LIN {X 0,Y 524.233,Z 362.321,A -85,B 0,C 180,E1 -4759.475,E2 -4759.475} C_VEL
LIN {X 0,Y 524.045,Z 370.841,A -85,B 0,C 180,E1 -4760.349,E2 -4760.349} C_VEL
LIN {X 0,Y 523.843,Z 378.7,A -85,B 0,C 180,E1 -4761.319,E2 -4761.319} C_VEL
LIN {X 0,Y 523.623,Z 386.372,A -85,B 0,C 180,E1 -4762.48,E2 -4762.48} C_VEL
LIN {X 0,Y 523.511,Z 393.443,A -85,B 0,C 180,E1 -4763.834,E2 -4763.834} C_VEL
LIN {X 0,Y 523.384,Z 398.145,A -85,B 0,C 180,E1 -4764.993,E2 -4764.993} C_VEL
LIN {X 0,Y 523.443,Z 401.738,A -85,B 0,C 180,E1 -4766.15,E2 -4766.15} C_VEL
LIN {X 0,Y 523.367,Z 403.59,A -85,B 0,C 180,E1 -4766.921,E2 -4766.921} C_VEL
LIN {X 0,Y 523.335,Z 404.979,A -85,B 0,C 180,E1 -4767.691,E2 -4767.691} C_VEL
LIN {X 0,Y 523.25,Z 406.574,A -85,B 0,C 180,E1 -4769.23,E2 -4769.23} C_VEL
LIN {X 0,Y 523.247,Z 406.79,A -85,B 0,C 180,E1 -4770,E2 -4770} C_VEL
LIN {X 0,Y 523.274,Z 405.972,A -85,B 0,C 180,E1 -4771.539,E2 -4771.539} C_VEL
LIN {X 0,Y 523.335,Z 404.983,A -85,B 0,C 180,E1 -4772.309,E2 -4772.309} C_VEL
LIN {X 0,Y 523.367,Z 403.595,A -85,B 0,C 180,E1 -4773.079,E2 -4773.079} C_VEL
LIN {X 0,Y 523.423,Z 400.675,A -85,B 0,C 180,E1 -4774.235,E2 -4774.235} C_VEL
LIN {X 0,Y 523.461,Z 396.72,A -85,B 0,C 180,E1 -4775.392,E2 -4775.392} C_VEL
LIN {X 0,Y 523.519,Z 391.508,A -85,B 0,C 180,E1 -4776.577,E2 -4776.577} C_VEL
LIN {X 0,Y 523.645,Z 385.219,A -85,B 0,C 180,E1 -4777.713,E2 -4777.713} C_VEL
LIN {X 0,Y 523.835,Z 377.219,A -85,B 0,C 180,E1 -4778.875,E2 -4778.875} C_VEL
LIN {X 0,Y 524.06,Z 369.064,A -85,B 0,C 180,E1 -4779.845,E2 -4779.845} C_VEL
LIN {X 0,Y 524.345,Z 359.117,A -85,B 0,C 180,E1 -4780.815,E2 -4780.815} C_VEL
LIN {X 0,Y 524.633,Z 347.823,A -85,B 0,C 180,E1 -4781.693,E2 -4781.693} C_VEL
LIN {X 0,Y 524.915,Z 336.875,A -85,B 0,C 180,E1 -4782.369,E2 -4782.369} C_VEL
LIN {X 0,Y 525.16,Z 324.67,A -85,B 0,C 180,E1 -4782.953,E2 -4782.953} C_VEL
LIN {X 0,Y 525.409,Z 311.875,A -85,B 0,C 180,E1 -4783.389,E2 -4783.389} C_VEL
LIN {X 0,Y 525.572,Z 298.314,A -85,B 0,C 180,E1 -4783.681,E2 -4783.681} C_VEL
LIN {X 0,Y 525.831,Z 204.563,A -85,B 0,C 180,E1 -4784.972,E2 -4784.972} C_VEL
LIN {X 0,Y 524.293,Z 195.105,A -85,B 0,C 180,E1 -4785.172,E2 -4785.172} C_VEL
LIN {X 0,Y 524.444,Z 184.228,A -85,B 0,C 180,E1 -4786.945,E2 -4786.945} C_VEL
LIN {X 0,Y 524.807,Z 168.725,A -85,B 0,C 180,E1 -4789.559,E2 -4789.559} C_VEL
LIN {X 0,Y 525.149,Z 155.599,A -85,B 0,C 180,E1 -4791.799,E2 -4791.799} C_VEL
LIN {X 0,Y 523.95,Z 148.335,A -85,B 0,C 180,E1 -4793.152,E2 -4793.152} C_VEL
LIN {X 0,Y 523.928,Z 148.217,A -85,B 0,C 180,E1 -4796.273,E2 -4796.273} C_VEL
LIN {X 0,Y 523.949,Z 148.223,A -85,B 0,C 180,E1 -4799.322,E2 -4799.322} C_VEL
LIN {X 0,Y 523.929,Z 148.219,A -85,B 0,C 180,E1 -4802.449,E2 -4802.449} C_VEL
LIN {X 0,Y 523.913,Z 148.227,A -85,B 0,C 180,E1 -4805.226,E2 -4805.226} C_VEL
LIN {X 0,Y 523.908,Z 148.214,A -85,B 0,C 180,E1 -4808.101,E2 -4808.101} C_VEL
LIN {X 0,Y 523.912,Z 148.228,A -85,B 0,C 180,E1 -4811.093,E2 -4811.093} C_VEL
LIN {X 0,Y 523.927,Z 148.218,A -85,B 0,C 180,E1 -4814.228,E2 -4814.228} C_VEL
LIN {X 0,Y 523.909,Z 148.224,A -85,B 0,C 180,E1 -4816.832,E2 -4816.832} C_VEL
LIN {X 0,Y 523.93,Z 148.224,A -85,B 0,C 180,E1 -4818.907,E2 -4818.907} C_VEL
LIN {X 0,Y 523.905,Z 148.215,A -85,B 0,C 180,E1 -4821.897,E2 -4821.897} C_VEL
LIN {X 0,Y 523.919,Z 148.218,A -85,B 0,C 180,E1 -4824.91,E2 -4824.91} C_VEL
LIN {X 0,Y 523.924,Z 148.219,A -85,B 0,C 180,E1 -4827.679,E2 -4827.679} C_VEL
LIN {X 0,Y 523.941,Z 148.22,A -85,B 0,C 180,E1 -4830.676,E2 -4830.676} C_VEL
LIN {X 0,Y 523.961,Z 148.213,A -85,B 0,C 180,E1 -4833.728,E2 -4833.728} C_VEL
LIN {X 0,Y 523.9,Z 148.219,A -85,B 0,C 180,E1 -4836.269,E2 -4836.269} C_VEL
LIN {X 0,Y 523.933,Z 148.225,A -85,B 0,C 180,E1 -4838.766,E2 -4838.766} C_VEL
LIN {X 0,Y 523.937,Z 148.215,A -85,B 0,C 180,E1 -4841.22,E2 -4841.22} C_VEL
LIN {X 0,Y 523.918,Z 148.217,A -85,B 0,C 180,E1 -4843.638,E2 -4843.638} C_VEL
LIN {X 0,Y 523.924,Z 148.219,A -85,B 0,C 180,E1 -4846.028,E2 -4846.028} C_VEL
LIN {X 0,Y 524,Z 148.208,A -85,B 0,C 180,E1 -4849.177,E2 -4849.177} C_VEL
LIN {X 0,Y 524.013,Z 148.211,A -85,B 0,C 180,E1 -4852.292,E2 -4852.292} C_VEL
LIN {X 0,Y 524.066,Z 148.203,A -85,B 0,C 180,E1 -4854.614,E2 -4854.614} C_VEL
LIN {X 0,Y 524.093,Z 148.196,A -85,B 0,C 180,E1 -4857.694,E2 -4857.694} C_VEL
LIN {X 0,Y 524.113,Z 148.196,A -85,B 0,C 180,E1 -4860.768,E2 -4860.768} C_VEL
LIN {X 0,Y 524.059,Z 148.2,A -85,B 0,C 180,E1 -4863.075,E2 -4863.075} C_VEL
LIN {X 0,Y 524.022,Z 148.21,A -85,B 0,C 180,E1 -4866.159,E2 -4866.159} C_VEL
LIN {X 0,Y 523.991,Z 148.212,A -85,B 0,C 180,E1 -4868.484,E2 -4868.484} C_VEL
LIN {X 0,Y 523.991,Z 148.21,A -85,B 0,C 180,E1 -4871.741,E2 -4871.741} C_VEL
LIN {X 0,Y 523.98,Z 148.208,A -85,B 0,C 180,E1 -4875.053,E2 -4875.053} C_VEL
LIN {X 0,Y 523.952,Z 148.217,A -85,B 0,C 180,E1 -4877.97,E2 -4877.97} C_VEL
LIN {X 0,Y 523.961,Z 148.218,A -85,B 0,C 180,E1 -4880.411,E2 -4880.411} C_VEL
LIN {X 0,Y 523.908,Z 148.219,A -85,B 0,C 180,E1 -4882.894,E2 -4882.894} C_VEL
LIN {X 0,Y 523.941,Z 148.216,A -85,B 0,C 180,E1 -4885.419,E2 -4885.419} C_VEL
LIN {X 0,Y 523.96,Z 148.218,A -85,B 0,C 180,E1 -4888,E2 -4888} C_VEL
LIN {X 0,Y 523.934,Z 148.217,A -85,B 0,C 180,E1 -4890.856,E2 -4890.856} C_VEL
LIN {X 0,Y 523.951,Z 148.215,A -85,B 0,C 180,E1 -4893.736,E2 -4893.736} C_VEL
LIN {X 0,Y 523.911,Z 148.219,A -85,B 0,C 180,E1 -4896.405,E2 -4896.405} C_VEL
LIN {X 0,Y 523.912,Z 148.219,A -85,B 0,C 180,E1 -4899.086,E2 -4899.086} C_VEL
LIN {X 0,Y 523.949,Z 148.215,A -85,B 0,C 180,E1 -4902.119,E2 -4902.119} C_VEL
LIN {X 0,Y 523.937,Z 148.215,A -85,B 0,C 180,E1 -4905.311,E2 -4905.311} C_VEL
LIN {X 0,Y 523.909,Z 148.22,A -85,B 0,C 180,E1 -4906.932,E2 -4906.932} C_VEL
LIN {X 0,Y 523.246,Z 148.308,A -85,B 0,C 180,E1 -4907.574,E2 -4907.574} C_VEL
LIN {X 0,Y 520.405,Z 148.661,A -85,B 0,C 180,E1 -4908.616,E2 -4908.616} C_VEL
LIN {X 0,Y 517.999,Z 148.961,A -85,B 0,C 180,E1 -4909.455,E2 -4909.455} C_VEL
LIN {X 0,Y 516.962,Z 149.086,A -85,B 0,C 180,E1 -4910.103,E2 -4910.103} C_VEL
LIN {X 0,Y 516.875,Z 149.095,A -85,B 0,C 180,E1 -4910.322,E2 -4910.322} C_VEL
LIN {X 0,Y 516.88,Z 149.099,A -85,B 0,C 180,E1 -4913.343,E2 -4913.343} C_VEL
LIN {X 0,Y 516.906,Z 149.097,A -85,B 0,C 180,E1 -4916.122,E2 -4916.122} C_VEL
LIN {X 0,Y 516.889,Z 149.092,A -85,B 0,C 180,E1 -4918.937,E2 -4918.937} C_VEL
LIN {X 0,Y 516.913,Z 149.097,A -85,B 0,C 180,E1 -4921.586,E2 -4921.586} C_VEL
LIN {X 0,Y 516.93,Z 149.094,A -85,B 0,C 180,E1 -4924.212,E2 -4924.212} C_VEL
LIN {X 0,Y 516.864,Z 149.1,A -85,B 0,C 180,E1 -4926.777,E2 -4926.777} C_VEL
LIN {X 0,Y 516.939,Z 149.232,A -85,B 0,C 180,E1 -4927.941,E2 -4927.941} C_VEL
LIN {X 0,Y 517.996,Z 155.265,A -85,B 0,C 180,E1 -4929.137,E2 -4929.137} C_VEL
LIN {X 0,Y 517.558,Z 172.414,A -85,B 0,C 180,E1 -4932.255,E2 -4932.255} C_VEL
LIN {X 0,Y 517.271,Z 186.072,A -85,B 0,C 180,E1 -4934.653,E2 -4934.653} C_VEL
LIN {X 0,Y 518.215,Z 191.523,A -85,B 0,C 180,E1 -4934.794,E2 -4934.794} C_VEL
LIN {X 0,Y 519.063,Z 197.009,A -85,B 0,C 180,E1 -4934.897,E2 -4934.897} C_VEL
LIN {X 0,Y 518.725,Z 293.597,A -85,B 0,C 180,E1 -4936.26,E2 -4936.26} C_VEL
LIN {X 0,Y 518.491,Z 306.768,A -85,B 0,C 180,E1 -4936.603,E2 -4936.603} C_VEL
LIN {X 0,Y 518.181,Z 318.87,A -85,B 0,C 180,E1 -4937.069,E2 -4937.069} C_VEL
LIN {X 0,Y 517.963,Z 330.449,A -85,B 0,C 180,E1 -4937.671,E2 -4937.671} C_VEL
LIN {X 0,Y 517.645,Z 341.982,A -85,B 0,C 180,E1 -4938.449,E2 -4938.449} C_VEL
LIN {X 0,Y 517.312,Z 352.479,A -85,B 0,C 180,E1 -4939.333,E2 -4939.333} C_VEL
LIN {X 0,Y 517.068,Z 361.057,A -85,B 0,C 180,E1 -4940.219,E2 -4940.219} C_VEL
LIN {X 0,Y 516.843,Z 368.96,A -85,B 0,C 180,E1 -4941.201,E2 -4941.201} C_VEL
LIN {X 0,Y 516.608,Z 376.691,A -85,B 0,C 180,E1 -4942.378,E2 -4942.378} C_VEL
LIN {X 0,Y 516.467,Z 383.782,A -85,B 0,C 180,E1 -4943.751,E2 -4943.751} C_VEL
LIN {X 0,Y 516.314,Z 388.51,A -85,B 0,C 180,E1 -4944.924,E2 -4944.924} C_VEL
LIN {X 0,Y 516.373,Z 392.131,A -85,B 0,C 180,E1 -4946.098,E2 -4946.098} C_VEL
LIN {X 0,Y 516.303,Z 394.004,A -85,B 0,C 180,E1 -4946.879,E2 -4946.879} C_VEL
LIN {X 0,Y 516.264,Z 395.418,A -85,B 0,C 180,E1 -4947.66,E2 -4947.66} C_VEL
LIN {X 0,Y 516.161,Z 397.042,A -85,B 0,C 180,E1 -4949.22,E2 -4949.22} C_VEL
LIN {X 0,Y 516.155,Z 397.28,A -85,B 0,C 180,E1 -4950,E2 -4950} C_VEL
LIN {X 0,Y 516.16,Z 397.096,A -85,B 0,C 180,E1 -4950.78,E2 -4950.78} C_VEL
LIN {X 0,Y 516.264,Z 395.543,A -85,B 0,C 180,E1 -4952.341,E2 -4952.341} C_VEL
LIN {X 0,Y 516.304,Z 394.184,A -85,B 0,C 180,E1 -4953.121,E2 -4953.121} C_VEL
LIN {X 0,Y 516.346,Z 391.311,A -85,B 0,C 180,E1 -4954.293,E2 -4954.293} C_VEL
LIN {X 0,Y 516.406,Z 387.415,A -85,B 0,C 180,E1 -4955.467,E2 -4955.467} C_VEL
LIN {X 0,Y 516.497,Z 381.513,A -85,B 0,C 180,E1 -4956.82,E2 -4956.82} C_VEL
LIN {X 0,Y 516.646,Z 374.84,A -85,B 0,C 180,E1 -4958.015,E2 -4958.015} C_VEL
LIN {X 0,Y 516.873,Z 366.667,A -85,B 0,C 180,E1 -4959.193,E2 -4959.193} C_VEL
LIN {X 0,Y 517.098,Z 358.304,A -85,B 0,C 180,E1 -4960.177,E2 -4960.177} C_VEL
LIN {X 0,Y 517.465,Z 347.982,A -85,B 0,C 180,E1 -4961.159,E2 -4961.159} C_VEL
LIN {X 0,Y 517.755,Z 336.363,A -85,B 0,C 180,E1 -4962.044,E2 -4962.044} C_VEL
LIN {X 0,Y 518.092,Z 324.766,A -85,B 0,C 180,E1 -4962.735,E2 -4962.735} C_VEL
LIN {X 0,Y 518.347,Z 312.735,A -85,B 0,C 180,E1 -4963.276,E2 -4963.276} C_VEL
LIN {X 0,Y 518.585,Z 299.648,A -85,B 0,C 180,E1 -4963.694,E2 -4963.694} C_VEL
LIN {X 0,Y 518.735,Z 287.139,A -85,B 0,C 180,E1 -4963.94,E2 -4963.94} C_VEL
LIN {X 0,Y 518.951,Z 195.763,A -85,B 0,C 180,E1 -4965.214,E2 -4965.214} C_VEL
LIN {X 0,Y 517.275,Z 186.34,A -85,B 0,C 180,E1 -4965.418,E2 -4965.418} C_VEL
LIN {X 0,Y 517.269,Z 184.001,A -85,B 0,C 180,E1 -4965.767,E2 -4965.767} C_VEL
LIN {X 0,Y 517.718,Z 165.889,A -85,B 0,C 180,E1 -4969.014,E2 -4969.014} C_VEL
LIN {X 0,Y 517.938,Z 154.621,A -85,B 0,C 180,E1 -4971.074,E2 -4971.074} C_VEL
LIN {X 0,Y 516.905,Z 149.156,A -85,B 0,C 180,E1 -4972.183,E2 -4972.183} C_VEL
LIN {X 0,Y 516.911,Z 149.097,A -85,B 0,C 180,E1 -4974.928,E2 -4974.928} C_VEL
LIN {X 0,Y 516.923,Z 149.095,A -85,B 0,C 180,E1 -4977.904,E2 -4977.904} C_VEL
LIN {X 0,Y 516.893,Z 149.102,A -85,B 0,C 180,E1 -4980.203,E2 -4980.203} C_VEL
LIN {X 0,Y 516.895,Z 149.096,A -85,B 0,C 180,E1 -4982.946,E2 -4982.946} C_VEL
LIN {X 0,Y 516.887,Z 149.093,A -85,B 0,C 180,E1 -4985.778,E2 -4985.778} C_VEL
LIN {X 0,Y 516.879,Z 149.094,A -85,B 0,C 180,E1 -4988.715,E2 -4988.715} C_VEL
LIN {X 0,Y 516.912,Z 149.091,A -85,B 0,C 180,E1 -4991.774,E2 -4991.774} C_VEL
LIN {X 0,Y 516.893,Z 149.091,A -85,B 0,C 180,E1 -4995.006,E2 -4995.006} C_VEL
LIN {X 0,Y 516.913,Z 149.095,A -85,B 0,C 180,E1 -4998.398,E2 -4998.398} C_VEL
LIN {X 0,Y 516.877,Z 149.096,A -85,B 0,C 180,E1 -5001.283,E2 -5001.283} C_VEL
LIN {X 0,Y 516.883,Z 149.087,A -85,B 0,C 180,E1 -5004.22,E2 -5004.22} C_VEL
LIN {X 0,Y 516.89,Z 149.09,A -85,B 0,C 180,E1 -5007.052,E2 -5007.052} C_VEL
LIN {X 0,Y 516.887,Z 149.101,A -85,B 0,C 180,E1 -5009.796,E2 -5009.796} C_VEL
LIN {X 0,Y 516.923,Z 149.089,A -85,B 0,C 180,E1 -5012.467,E2 -5012.467} C_VEL
LIN {X 0,Y 516.866,Z 149.098,A -85,B 0,C 180,E1 -5015.069,E2 -5015.069} C_VEL
LIN {X 0,Y 516.862,Z 149.102,A -85,B 0,C 180,E1 -5017.621,E2 -5017.621} C_VEL
LIN {X 0,Y 516.924,Z 149.094,A -85,B 0,C 180,E1 -5020.129,E2 -5020.129} C_VEL
LIN {X 0,Y 516.914,Z 149.09,A -85,B 0,C 180,E1 -5022.596,E2 -5022.596} C_VEL
LIN {X 0,Y 516.935,Z 149.085,A -85,B 0,C 180,E1 -5025.03,E2 -5025.03} C_VEL
LIN {X 0,Y 516.958,Z 149.086,A -85,B 0,C 180,E1 -5028.233,E2 -5028.233} C_VEL
LIN {X 0,Y 516.961,Z 149.085,A -85,B 0,C 180,E1 -5031.399,E2 -5031.399} C_VEL
LIN {X 0,Y 516.992,Z 149.088,A -85,B 0,C 180,E1 -5033.757,E2 -5033.757} C_VEL
LIN {X 0,Y 517.003,Z 149.078,A -85,B 0,C 180,E1 -5036.883,E2 -5036.883} C_VEL
LIN {X 0,Y 517.072,Z 149.074,A -85,B 0,C 180,E1 -5040,E2 -5040} C_VEL
LIN {X 0,Y 517.004,Z 149.083,A -85,B 0,C 180,E1 -5043.117,E2 -5043.117} C_VEL
LIN {X 0,Y 516.993,Z 149.08,A -85,B 0,C 180,E1 -5046.243,E2 -5046.243} C_VEL
LIN {X 0,Y 516.939,Z 149.095,A -85,B 0,C 180,E1 -5049.389,E2 -5049.389} C_VEL
LIN {X 0,Y 516.944,Z 149.087,A -85,B 0,C 180,E1 -5051.807,E2 -5051.807} C_VEL
LIN {X 0,Y 516.937,Z 149.095,A -85,B 0,C 180,E1 -5055.146,E2 -5055.146} C_VEL
LIN {X 0,Y 516.908,Z 149.088,A -85,B 0,C 180,E1 -5058.223,E2 -5058.223} C_VEL
LIN {X 0,Y 516.898,Z 149.095,A -85,B 0,C 180,E1 -5060.702,E2 -5060.702} C_VEL
LIN {X 0,Y 516.883,Z 149.092,A -85,B 0,C 180,E1 -5064.073,E2 -5064.073} C_VEL
LIN {X 0,Y 516.917,Z 149.093,A -85,B 0,C 180,E1 -5066.658,E2 -5066.658} C_VEL
LIN {X 0,Y 516.902,Z 149.094,A -85,B 0,C 180,E1 -5069.524,E2 -5069.524} C_VEL
LIN {X 0,Y 516.888,Z 149.097,A -85,B 0,C 180,E1 -5072.543,E2 -5072.543} C_VEL
LIN {X 0,Y 516.86,Z 149.092,A -85,B 0,C 180,E1 -5075.33,E2 -5075.33} C_VEL
LIN {X 0,Y 516.874,Z 149.091,A -85,B 0,C 180,E1 -5077.943,E2 -5077.943} C_VEL
LIN {X 0,Y 516.878,Z 149.101,A -85,B 0,C 180,E1 -5080.742,E2 -5080.742} C_VEL
LIN {X 0,Y 516.877,Z 149.095,A -85,B 0,C 180,E1 -5083.904,E2 -5083.904} C_VEL
LIN {X 0,Y 516.878,Z 149.096,A -85,B 0,C 180,E1 -5086.108,E2 -5086.108} C_VEL
LIN {X 0,Y 516.859,Z 149.101,A -85,B 0,C 180,E1 -5089.257,E2 -5089.257} C_VEL
LIN {X 0,Y 516.876,Z 149.091,A -85,B 0,C 180,E1 -5092.058,E2 -5092.058} C_VEL
LIN {X 0,Y 516.88,Z 149.096,A -85,B 0,C 180,E1 -5095.176,E2 -5095.176} C_VEL
LIN {X 0,Y 516.872,Z 149.098,A -85,B 0,C 180,E1 -5097.975,E2 -5097.975} C_VEL
LIN {X 0,Y 516.919,Z 149.099,A -85,B 0,C 180,E1 -5100.696,E2 -5100.696} C_VEL
LIN {X 0,Y 516.896,Z 149.094,A -85,B 0,C 180,E1 -5103.815,E2 -5103.815} C_VEL
LIN {X 0,Y 516.895,Z 149.193,A -85,B 0,C 180,E1 -5106.672,E2 -5106.672} C_VEL
LIN {X 0,Y 518.203,Z 156.728,A -85,B 0,C 180,E1 -5108.102,E2 -5108.102} C_VEL
LIN {X 0,Y 517.794,Z 173.43,A -85,B 0,C 180,E1 -5110.989,E2 -5110.989} C_VEL
LIN {X 0,Y 517.328,Z 191.313,A -85,B 0,C 180,E1 -5114.032,E2 -5114.032} C_VEL
LIN {X 0,Y 517.292,Z 195.135,A -85,B 0,C 180,E1 -5114.623,E2 -5114.623} C_VEL
LIN {X 0,Y 519.102,Z 207.405,A -85,B 0,C 180,E1 -5114.87,E2 -5114.87} C_VEL
LIN {X 0,Y 518.674,Z 302.556,A -85,B 0,C 180,E1 -5116.208,E2 -5116.208} C_VEL
LIN {X 0,Y 518.41,Z 315.831,A -85,B 0,C 180,E1 -5116.551,E2 -5116.551} C_VEL
LIN {X 0,Y 518.138,Z 329.11,A -85,B 0,C 180,E1 -5117.067,E2 -5117.067} C_VEL
LIN {X 0,Y 517.837,Z 341.482,A -85,B 0,C 180,E1 -5117.735,E2 -5117.735} C_VEL
LIN {X 0,Y 517.536,Z 353.125,A -85,B 0,C 180,E1 -5118.545,E2 -5118.545} C_VEL
LIN {X 0,Y 517.222,Z 363.299,A -85,B 0,C 180,E1 -5119.43,E2 -5119.43} C_VEL
LIN {X 0,Y 516.956,Z 372.45,A -85,B 0,C 180,E1 -5120.413,E2 -5120.413} C_VEL
LIN {X 0,Y 516.71,Z 381.365,A -85,B 0,C 180,E1 -5121.592,E2 -5121.592} C_VEL
LIN {X 0,Y 516.505,Z 388.538,A -85,B 0,C 180,E1 -5122.769,E2 -5122.769} C_VEL
LIN {X 0,Y 516.427,Z 395.068,A -85,B 0,C 180,E1 -5124.142,E2 -5124.142} C_VEL
LIN {X 0,Y 516.269,Z 399.386,A -85,B 0,C 180,E1 -5125.315,E2 -5125.315} C_VEL
LIN {X 0,Y 516.352,Z 401.673,A -85,B 0,C 180,E1 -5126.098,E2 -5126.098} C_VEL
LIN {X 0,Y 516.282,Z 403.525,A -85,B 0,C 180,E1 -5126.878,E2 -5126.878} C_VEL
LIN {X 0,Y 516.261,Z 404.914,A -85,B 0,C 180,E1 -5127.659,E2 -5127.659} C_VEL
LIN {X 0,Y 516.16,Z 406.509,A -85,B 0,C 180,E1 -5129.22,E2 -5129.22} C_VEL
LIN {X 0,Y 516.154,Z 406.725,A -85,B 0,C 180,E1 -5130,E2 -5130} C_VEL
LIN {X 0,Y 516.192,Z 405.907,A -85,B 0,C 180,E1 -5131.56,E2 -5131.56} C_VEL
LIN {X 0,Y 516.261,Z 404.918,A -85,B 0,C 180,E1 -5132.34,E2 -5132.34} C_VEL
LIN {X 0,Y 516.282,Z 403.53,A -85,B 0,C 180,E1 -5133.121,E2 -5133.121} C_VEL
LIN {X 0,Y 516.312,Z 400.609,A -85,B 0,C 180,E1 -5134.293,E2 -5134.293} C_VEL
LIN {X 0,Y 516.397,Z 396.655,A -85,B 0,C 180,E1 -5135.466,E2 -5135.466} C_VEL
LIN {X 0,Y 516.478,Z 390.787,A -85,B 0,C 180,E1 -5136.796,E2 -5136.796} C_VEL
LIN {X 0,Y 516.628,Z 383.921,A -85,B 0,C 180,E1 -5138.015,E2 -5138.015} C_VEL
LIN {X 0,Y 516.843,Z 375.667,A -85,B 0,C 180,E1 -5139.193,E2 -5139.193} C_VEL
LIN {X 0,Y 517.064,Z 367.204,A -85,B 0,C 180,E1 -5140.177,E2 -5140.177} C_VEL
LIN {X 0,Y 517.411,Z 356.744,A -85,B 0,C 180,E1 -5141.16,E2 -5141.16} C_VEL
LIN {X 0,Y 517.727,Z 345.028,A -85,B 0,C 180,E1 -5142.042,E2 -5142.042} C_VEL
LIN {X 0,Y 518.054,Z 333.123,A -85,B 0,C 180,E1 -5142.735,E2 -5142.735} C_VEL
LIN {X 0,Y 518.325,Z 320.798,A -85,B 0,C 180,E1 -5143.276,E2 -5143.276} C_VEL
LIN {X 0,Y 518.559,Z 308.151,A -85,B 0,C 180,E1 -5143.669,E2 -5143.669} C_VEL
LIN {X 0,Y 518.749,Z 294.967,A -85,B 0,C 180,E1 -5143.914,E2 -5143.914} C_VEL
LIN {X 0,Y 519.051,Z 206.099,A -85,B 0,C 180,E1 -5145.15,E2 -5145.15} C_VEL
LIN {X 0,Y 517.298,Z 195.066,A -85,B 0,C 180,E1 -5145.38,E2 -5145.38} C_VEL
LIN {X 0,Y 517.562,Z 181.901,A -85,B 0,C 180,E1 -5147.564,E2 -5147.564} C_VEL
LIN {X 0,Y 518.054,Z 163.89,A -85,B 0,C 180,E1 -5150.653,E2 -5150.653} C_VEL
LIN {X 0,Y 518.099,Z 155.533,A -85,B 0,C 180,E1 -5152.112,E2 -5152.112} C_VEL
LIN {X 0,Y 516.894,Z 149.193,A -85,B 0,C 180,E1 -5153.327,E2 -5153.327} C_VEL
LIN {X 0,Y 516.892,Z 149.091,A -85,B 0,C 180,E1 -5156.659,E2 -5156.659} C_VEL
LIN {X 0,Y 516.904,Z 149.097,A -85,B 0,C 180,E1 -5159.522,E2 -5159.522} C_VEL
LIN {X 0,Y 516.892,Z 149.096,A -85,B 0,C 180,E1 -5162.542,E2 -5162.542} C_VEL
LIN {X 0,Y 516.859,Z 149.106,A -85,B 0,C 180,E1 -5165.328,E2 -5165.328} C_VEL
LIN {X 0,Y 516.873,Z 149.091,A -85,B 0,C 180,E1 -5167.942,E2 -5167.942} C_VEL
LIN {X 0,Y 516.865,Z 149.1,A -85,B 0,C 180,E1 -5170.742,E2 -5170.742} C_VEL
LIN {X 0,Y 516.875,Z 149.096,A -85,B 0,C 180,E1 -5173.902,E2 -5173.902} C_VEL
LIN {X 0,Y 516.874,Z 149.095,A -85,B 0,C 180,E1 -5176.106,E2 -5176.106} C_VEL
LIN {X 0,Y 516.905,Z 149.093,A -85,B 0,C 180,E1 -5178.398,E2 -5178.398} C_VEL
LIN {X 0,Y 516.871,Z 149.095,A -85,B 0,C 180,E1 -5181.283,E2 -5181.283} C_VEL
LIN {X 0,Y 516.863,Z 149.088,A -85,B 0,C 180,E1 -5184.219,E2 -5184.219} C_VEL
LIN {X 0,Y 516.871,Z 149.104,A -85,B 0,C 180,E1 -5187.051,E2 -5187.051} C_VEL
LIN {X 0,Y 516.875,Z 149.094,A -85,B 0,C 180,E1 -5189.795,E2 -5189.795} C_VEL
LIN {X 0,Y 516.912,Z 149.094,A -85,B 0,C 180,E1 -5192.466,E2 -5192.466} C_VEL
LIN {X 0,Y 516.86,Z 149.099,A -85,B 0,C 180,E1 -5195.069,E2 -5195.069} C_VEL
LIN {X 0,Y 516.856,Z 149.098,A -85,B 0,C 180,E1 -5197.621,E2 -5197.621} C_VEL
LIN {X 0,Y 516.919,Z 149.091,A -85,B 0,C 180,E1 -5200.129,E2 -5200.129} C_VEL
LIN {X 0,Y 516.894,Z 149.096,A -85,B 0,C 180,E1 -5202.595,E2 -5202.595} C_VEL
LIN {X 0,Y 516.929,Z 149.094,A -85,B 0,C 180,E1 -5205.03,E2 -5205.03} C_VEL
LIN {X 0,Y 516.991,Z 149.081,A -85,B 0,C 180,E1 -5208.234,E2 -5208.234} C_VEL
LIN {X 0,Y 516.951,Z 149.087,A -85,B 0,C 180,E1 -5211.399,E2 -5211.399} C_VEL
LIN {X 0,Y 516.988,Z 149.081,A -85,B 0,C 180,E1 -5213.757,E2 -5213.757} C_VEL
LIN {X 0,Y 517,Z 149.084,A -85,B 0,C 180,E1 -5216.883,E2 -5216.883} C_VEL
LIN {X 0,Y 517.066,Z 149.074,A -85,B 0,C 180,E1 -5220,E2 -5220} C_VEL
LIN {X 0,Y 517,Z 149.078,A -85,B 0,C 180,E1 -5223.117,E2 -5223.117} C_VEL
LIN {X 0,Y 516.987,Z 149.088,A -85,B 0,C 180,E1 -5226.244,E2 -5226.244} C_VEL
LIN {X 0,Y 516.94,Z 149.082,A -85,B 0,C 180,E1 -5229.39,E2 -5229.39} C_VEL
LIN {X 0,Y 516.94,Z 149.088,A -85,B 0,C 180,E1 -5231.808,E2 -5231.808} C_VEL
LIN {X 0,Y 516.931,Z 149.085,A -85,B 0,C 180,E1 -5235.147,E2 -5235.147} C_VEL
LIN {X 0,Y 516.913,Z 149.098,A -85,B 0,C 180,E1 -5238.223,E2 -5238.223} C_VEL
LIN {X 0,Y 516.902,Z 149.093,A -85,B 0,C 180,E1 -5240.702,E2 -5240.702} C_VEL
LIN {X 0,Y 516.863,Z 149.096,A -85,B 0,C 180,E1 -5243.224,E2 -5243.224} C_VEL
LIN {X 0,Y 516.932,Z 149.096,A -85,B 0,C 180,E1 -5246.197,E2 -5246.197} C_VEL
LIN {X 0,Y 516.912,Z 149.091,A -85,B 0,C 180,E1 -5249.305,E2 -5249.305} C_VEL
LIN {X 0,Y 516.886,Z 149.093,A -85,B 0,C 180,E1 -5252.544,E2 -5252.544} C_VEL
LIN {X 0,Y 516.87,Z 149.084,A -85,B 0,C 180,E1 -5255.333,E2 -5255.333} C_VEL
LIN {X 0,Y 516.872,Z 149.1,A -85,B 0,C 180,E1 -5257.944,E2 -5257.944} C_VEL
LIN {X 0,Y 516.878,Z 149.095,A -85,B 0,C 180,E1 -5260.742,E2 -5260.742} C_VEL
LIN {X 0,Y 516.876,Z 149.088,A -85,B 0,C 180,E1 -5262.832,E2 -5262.832} C_VEL
LIN {X 0,Y 516.888,Z 149.091,A -85,B 0,C 180,E1 -5265.008,E2 -5265.008} C_VEL
LIN {X 0,Y 516.909,Z 149.091,A -85,B 0,C 180,E1 -5268.4,E2 -5268.4} C_VEL
LIN {X 0,Y 516.875,Z 149.095,A -85,B 0,C 180,E1 -5270.322,E2 -5270.322} C_VEL
LIN {X 0,Y 516.205,Z 149.177,A -85,B 0,C 180,E1 -5270.972,E2 -5270.972} C_VEL
LIN {X 0,Y 513.36,Z 149.541,A -85,B 0,C 180,E1 -5272.028,E2 -5272.028} C_VEL
LIN {X 0,Y 510.953,Z 149.846,A -85,B 0,C 180,E1 -5272.878,E2 -5272.878} C_VEL
LIN {X 0,Y 509.913,Z 149.972,A -85,B 0,C 180,E1 -5273.535,E2 -5273.535} C_VEL
LIN {X 0,Y 509.824,Z 149.979,A -85,B 0,C 180,E1 -5273.757,E2 -5273.757} C_VEL
LIN {X 0,Y 509.857,Z 149.972,A -85,B 0,C 180,E1 -5276.54,E2 -5276.54} C_VEL
LIN {X 0,Y 509.843,Z 149.972,A -85,B 0,C 180,E1 -5279.335,E2 -5279.335} C_VEL
LIN {X 0,Y 509.887,Z 149.973,A -85,B 0,C 180,E1 -5282.055,E2 -5282.055} C_VEL
LIN {X 0,Y 509.875,Z 149.971,A -85,B 0,C 180,E1 -5284.705,E2 -5284.705} C_VEL
LIN {X 0,Y 509.881,Z 150.069,A -85,B 0,C 180,E1 -5287.765,E2 -5287.765} C_VEL
LIN {X 0,Y 511.033,Z 156.403,A -85,B 0,C 180,E1 -5289.05,E2 -5289.05} C_VEL
LIN {X 0,Y 510.602,Z 172.735,A -85,B 0,C 180,E1 -5292.058,E2 -5292.058} C_VEL
LIN {X 0,Y 510.25,Z 186.058,A -85,B 0,C 180,E1 -5294.429,E2 -5294.429} C_VEL
LIN {X 0,Y 510.842,Z 189.565,A -85,B 0,C 180,E1 -5294.539,E2 -5294.539} C_VEL
LIN {X 0,Y 512.221,Z 197.251,A -85,B 0,C 180,E1 -5294.692,E2 -5294.692} C_VEL
LIN {X 0,Y 511.828,Z 293.69,A -85,B 0,C 180,E1 -5296.071,E2 -5296.071} C_VEL
LIN {X 0,Y 511.59,Z 306.852,A -85,B 0,C 180,E1 -5296.419,E2 -5296.419} C_VEL
LIN {X 0,Y 511.265,Z 318.949,A -85,B 0,C 180,E1 -5296.891,E2 -5296.891} C_VEL
LIN {X 0,Y 511.024,Z 330.472,A -85,B 0,C 180,E1 -5297.498,E2 -5297.498} C_VEL
LIN {X 0,Y 510.696,Z 342.055,A -85,B 0,C 180,E1 -5298.289,E2 -5298.289} C_VEL
LIN {X 0,Y 510.32,Z 352.551,A -85,B 0,C 180,E1 -5299.186,E2 -5299.186} C_VEL
LIN {X 0,Y 510.071,Z 361.128,A -85,B 0,C 180,E1 -5300.083,E2 -5300.083} C_VEL
LIN {X 0,Y 509.815,Z 369.03,A -85,B 0,C 180,E1 -5301.079,E2 -5301.079} C_VEL
LIN {X 0,Y 509.544,Z 376.759,A -85,B 0,C 180,E1 -5302.272,E2 -5302.272} C_VEL
LIN {X 0,Y 509.382,Z 383.85,A -85,B 0,C 180,E1 -5303.663,E2 -5303.663} C_VEL
LIN {X 0,Y 509.249,Z 388.578,A -85,B 0,C 180,E1 -5304.854,E2 -5304.854} C_VEL
LIN {X 0,Y 509.286,Z 392.198,A -85,B 0,C 180,E1 -5306.044,E2 -5306.044} C_VEL
LIN {X 0,Y 509.22,Z 394.07,A -85,B 0,C 180,E1 -5306.836,E2 -5306.836} C_VEL
LIN {X 0,Y 509.193,Z 395.483,A -85,B 0,C 180,E1 -5307.627,E2 -5307.627} C_VEL
LIN {X 0,Y 509.074,Z 397.107,A -85,B 0,C 180,E1 -5309.209,E2 -5309.209} C_VEL
LIN {X 0,Y 509.066,Z 397.345,A -85,B 0,C 180,E1 -5310,E2 -5310} C_VEL
LIN {X 0,Y 509.074,Z 397.161,A -85,B 0,C 180,E1 -5310.791,E2 -5310.791} C_VEL
LIN {X 0,Y 509.194,Z 395.607,A -85,B 0,C 180,E1 -5312.373,E2 -5312.373} C_VEL
LIN {X 0,Y 509.221,Z 394.247,A -85,B 0,C 180,E1 -5313.165,E2 -5313.165} C_VEL
LIN {X 0,Y 509.254,Z 391.374,A -85,B 0,C 180,E1 -5314.353,E2 -5314.353} C_VEL
LIN {X 0,Y 509.349,Z 387.477,A -85,B 0,C 180,E1 -5315.543,E2 -5315.543} C_VEL
LIN {X 0,Y 509.417,Z 382.453,A -85,B 0,C 180,E1 -5316.734,E2 -5316.734} C_VEL
LIN {X 0,Y 509.569,Z 376.127,A -85,B 0,C 180,E1 -5317.928,E2 -5317.928} C_VEL
LIN {X 0,Y 509.792,Z 368.21,A -85,B 0,C 180,E1 -5319.122,E2 -5319.122} C_VEL
LIN {X 0,Y 510.055,Z 360.142,A -85,B 0,C 180,E1 -5320.118,E2 -5320.118} C_VEL
LIN {X 0,Y 510.393,Z 350.298,A -85,B 0,C 180,E1 -5321.115,E2 -5321.115} C_VEL
LIN {X 0,Y 510.718,Z 340.618,A -85,B 0,C 180,E1 -5321.912,E2 -5321.912} C_VEL
LIN {X 0,Y 510.991,Z 329.744,A -85,B 0,C 180,E1 -5322.636,E2 -5322.636} C_VEL
LIN {X 0,Y 511.329,Z 317.565,A -85,B 0,C 180,E1 -5323.26,E2 -5323.26} C_VEL
LIN {X 0,Y 511.611,Z 304.21,A -85,B 0,C 180,E1 -5323.758,E2 -5323.758} C_VEL
LIN {X 0,Y 511.842,Z 291.733,A -85,B 0,C 180,E1 -5324.056,E2 -5324.056} C_VEL
LIN {X 0,Y 512.139,Z 196.775,A -85,B 0,C 180,E1 -5325.407,E2 -5325.407} C_VEL
LIN {X 0,Y 510.267,Z 186.28,A -85,B 0,C 180,E1 -5325.639,E2 -5325.639} C_VEL
LIN {X 0,Y 510.385,Z 180.631,A -85,B 0,C 180,E1 -5326.602,E2 -5326.602} C_VEL
LIN {X 0,Y 510.771,Z 164.778,A -85,B 0,C 180,E1 -5329.492,E2 -5329.492} C_VEL
LIN {X 0,Y 510.96,Z 155.754,A -85,B 0,C 180,E1 -5331.165,E2 -5331.165} C_VEL
LIN {X 0,Y 509.844,Z 150.035,A -85,B 0,C 180,E1 -5332.343,E2 -5332.343} C_VEL
LIN {X 0,Y 509.878,Z 149.971,A -85,B 0,C 180,E1 -5335.296,E2 -5335.296} C_VEL
LIN {X 0,Y 509.895,Z 149.972,A -85,B 0,C 180,E1 -5338.1,E2 -5338.1} C_VEL
LIN {X 0,Y 509.846,Z 149.968,A -85,B 0,C 180,E1 -5341.279,E2 -5341.279} C_VEL
LIN {X 0,Y 509.86,Z 149.974,A -85,B 0,C 180,E1 -5344.203,E2 -5344.203} C_VEL
LIN {X 0,Y 509.818,Z 149.976,A -85,B 0,C 180,E1 -5347.34,E2 -5347.34} C_VEL
LIN {X 0,Y 509.837,Z 149.973,A -85,B 0,C 180,E1 -5350.382,E2 -5350.382} C_VEL
LIN {X 0,Y 509.821,Z 149.975,A -85,B 0,C 180,E1 -5353.062,E2 -5353.062} C_VEL
LIN {X 0,Y 509.82,Z 149.976,A -85,B 0,C 180,E1 -5355.793,E2 -5355.793} C_VEL
LIN {X 0,Y 509.855,Z 149.972,A -85,B 0,C 180,E1 -5358.574,E2 -5358.574} C_VEL
LIN {X 0,Y 509.847,Z 149.977,A -85,B 0,C 180,E1 -5361.786,E2 -5361.786} C_VEL
LIN {X 0,Y 509.836,Z 149.959,A -85,B 0,C 180,E1 -5364.622,E2 -5364.622} C_VEL
LIN {X 0,Y 509.856,Z 149.968,A -85,B 0,C 180,E1 -5367.48,E2 -5367.48} C_VEL
LIN {X 0,Y 509.853,Z 149.974,A -85,B 0,C 180,E1 -5370.273,E2 -5370.273} C_VEL
LIN {X 0,Y 509.88,Z 149.964,A -85,B 0,C 180,E1 -5372.944,E2 -5372.944} C_VEL
LIN {X 0,Y 509.843,Z 149.977,A -85,B 0,C 180,E1 -5375.572,E2 -5375.572} C_VEL
LIN {X 0,Y 509.815,Z 149.977,A -85,B 0,C 180,E1 -5378.148,E2 -5378.148} C_VEL
LIN {X 0,Y 509.855,Z 149.971,A -85,B 0,C 180,E1 -5380.681,E2 -5380.681} C_VEL
LIN {X 0,Y 509.875,Z 149.968,A -85,B 0,C 180,E1 -5383.174,E2 -5383.174} C_VEL
LIN {X 0,Y 509.856,Z 149.973,A -85,B 0,C 180,E1 -5385.634,E2 -5385.634} C_VEL
LIN {X 0,Y 509.905,Z 149.963,A -85,B 0,C 180,E1 -5388.874,E2 -5388.874} C_VEL
LIN {X 0,Y 509.944,Z 149.961,A -85,B 0,C 180,E1 -5392.078,E2 -5392.078} C_VEL
LIN {X 0,Y 509.97,Z 149.956,A -85,B 0,C 180,E1 -5394.464,E2 -5394.464} C_VEL
LIN {X 0,Y 510.044,Z 149.949,A -85,B 0,C 180,E1 -5397.631,E2 -5397.631} C_VEL
LIN {X 0,Y 510.043,Z 149.95,A -85,B 0,C 180,E1 -5400,E2 -5400} C_VEL
LIN {X 0,Y 510.042,Z 149.946,A -85,B 0,C 180,E1 -5402.369,E2 -5402.369} C_VEL
LIN {X 0,Y 509.944,Z 149.958,A -85,B 0,C 180,E1 -5406.33,E2 -5406.33} C_VEL
LIN {X 0,Y 509.879,Z 149.972,A -85,B 0,C 180,E1 -5409.521,E2 -5409.521} C_VEL
LIN {X 0,Y 509.897,Z 149.964,A -85,B 0,C 180,E1 -5411.932,E2 -5411.932} C_VEL
LIN {X 0,Y 509.887,Z 149.974,A -85,B 0,C 180,E1 -5415.242,E2 -5415.242} C_VEL
LIN {X 0,Y 509.854,Z 149.967,A -85,B 0,C 180,E1 -5418.484,E2 -5418.484} C_VEL
LIN {X 0,Y 509.839,Z 149.978,A -85,B 0,C 180,E1 -5421.002,E2 -5421.002} C_VEL
LIN {X 0,Y 509.815,Z 149.976,A -85,B 0,C 180,E1 -5423.564,E2 -5423.564} C_VEL
LIN {X 0,Y 509.904,Z 149.965,A -85,B 0,C 180,E1 -5426.379,E2 -5426.379} C_VEL
LIN {X 0,Y 509.866,Z 149.973,A -85,B 0,C 180,E1 -5428.845,E2 -5428.845} C_VEL
LIN {X 0,Y 509.813,Z 149.979,A -85,B 0,C 180,E1 -5431.591,E2 -5431.591} C_VEL
LIN {X 0,Y 509.833,Z 149.972,A -85,B 0,C 180,E1 -5434.415,E2 -5434.415} C_VEL
LIN {X 0,Y 509.811,Z 149.974,A -85,B 0,C 180,E1 -5437.341,E2 -5437.341} C_VEL
LIN {X 0,Y 509.834,Z 149.974,A -85,B 0,C 180,E1 -5440.383,E2 -5440.383} C_VEL
LIN {X 0,Y 509.797,Z 149.982,A -85,B 0,C 180,E1 -5443.06,E2 -5443.06} C_VEL
LIN {X 0,Y 509.819,Z 149.975,A -85,B 0,C 180,E1 -5445.794,E2 -5445.794} C_VEL
LIN {X 0,Y 509.83,Z 149.978,A -85,B 0,C 180,E1 -5448.573,E2 -5448.573} C_VEL
LIN {X 0,Y 509.848,Z 149.965,A -85,B 0,C 180,E1 -5451.787,E2 -5451.787} C_VEL
LIN {X 0,Y 509.826,Z 149.982,A -85,B 0,C 180,E1 -5454.622,E2 -5454.622} C_VEL
LIN {X 0,Y 509.86,Z 149.972,A -85,B 0,C 180,E1 -5457.481,E2 -5457.481} C_VEL
LIN {X 0,Y 509.858,Z 149.973,A -85,B 0,C 180,E1 -5460.274,E2 -5460.274} C_VEL
LIN {X 0,Y 509.858,Z 149.965,A -85,B 0,C 180,E1 -5462.943,E2 -5462.943} C_VEL
LIN {X 0,Y 509.867,Z 150.052,A -85,B 0,C 180,E1 -5466.492,E2 -5466.492} C_VEL
LIN {X 0,Y 511.128,Z 156.665,A -85,B 0,C 180,E1 -5467.783,E2 -5467.783} C_VEL
LIN {X 0,Y 511.016,Z 166.762,A -85,B 0,C 180,E1 -5469.567,E2 -5469.567} C_VEL
LIN {X 0,Y 510.556,Z 182.906,A -85,B 0,C 180,E1 -5472.372,E2 -5472.372} C_VEL
LIN {X 0,Y 510.271,Z 194.938,A -85,B 0,C 180,E1 -5474.398,E2 -5474.398} C_VEL
LIN {X 0,Y 512.252,Z 207.254,A -85,B 0,C 180,E1 -5474.662,E2 -5474.662} C_VEL
LIN {X 0,Y 511.799,Z 302.491,A -85,B 0,C 180,E1 -5476.019,E2 -5476.019} C_VEL
LIN {X 0,Y 511.491,Z 315.766,A -85,B 0,C 180,E1 -5476.365,E2 -5476.365} C_VEL
LIN {X 0,Y 511.196,Z 329.045,A -85,B 0,C 180,E1 -5476.889,E2 -5476.889} C_VEL
LIN {X 0,Y 510.877,Z 341.412,A -85,B 0,C 180,E1 -5477.565,E2 -5477.565} C_VEL
LIN {X 0,Y 510.576,Z 353.06,A -85,B 0,C 180,E1 -5478.386,E2 -5478.386} C_VEL
LIN {X 0,Y 510.196,Z 363.233,A -85,B 0,C 180,E1 -5479.283,E2 -5479.283} C_VEL
LIN {X 0,Y 509.946,Z 372.385,A -85,B 0,C 180,E1 -5480.28,E2 -5480.28} C_VEL
LIN {X 0,Y 509.652,Z 381.3,A -85,B 0,C 180,E1 -5481.475,E2 -5481.475} C_VEL
LIN {X 0,Y 509.433,Z 388.473,A -85,B 0,C 180,E1 -5482.668,E2 -5482.668} C_VEL
LIN {X 0,Y 509.32,Z 393.312,A -85,B 0,C 180,E1 -5483.662,E2 -5483.662} C_VEL
LIN {X 0,Y 509.246,Z 398.015,A -85,B 0,C 180,E1 -5484.853,E2 -5484.853} C_VEL
LIN {X 0,Y 509.246,Z 401.608,A -85,B 0,C 180,E1 -5486.043,E2 -5486.043} C_VEL
LIN {X 0,Y 509.2,Z 403.46,A -85,B 0,C 180,E1 -5486.835,E2 -5486.835} C_VEL
LIN {X 0,Y 509.161,Z 404.849,A -85,B 0,C 180,E1 -5487.626,E2 -5487.626} C_VEL
LIN {X 0,Y 509.073,Z 406.445,A -85,B 0,C 180,E1 -5489.209,E2 -5489.209} C_VEL
LIN {X 0,Y 509.066,Z 406.66,A -85,B 0,C 180,E1 -5490,E2 -5490} C_VEL
LIN {X 0,Y 509.112,Z 405.842,A -85,B 0,C 180,E1 -5491.582,E2 -5491.582} C_VEL
LIN {X 0,Y 509.161,Z 404.853,A -85,B 0,C 180,E1 -5492.373,E2 -5492.373} C_VEL
LIN {X 0,Y 509.2,Z 403.465,A -85,B 0,C 180,E1 -5493.164,E2 -5493.164} C_VEL
LIN {X 0,Y 509.206,Z 400.544,A -85,B 0,C 180,E1 -5494.353,E2 -5494.353} C_VEL
LIN {X 0,Y 509.311,Z 396.59,A -85,B 0,C 180,E1 -5495.543,E2 -5495.543} C_VEL
LIN {X 0,Y 509.401,Z 390.959,A -85,B 0,C 180,E1 -5496.844,E2 -5496.844} C_VEL
LIN {X 0,Y 509.562,Z 383.856,A -85,B 0,C 180,E1 -5498.127,E2 -5498.127} C_VEL
LIN {X 0,Y 509.803,Z 375.601,A -85,B 0,C 180,E1 -5499.321,E2 -5499.321} C_VEL
LIN {X 0,Y 510.051,Z 367.139,A -85,B 0,C 180,E1 -5500.318,E2 -5500.318} C_VEL
LIN {X 0,Y 510.433,Z 356.679,A -85,B 0,C 180,E1 -5501.314,E2 -5501.314} C_VEL
LIN {X 0,Y 510.743,Z 345.832,A -85,B 0,C 180,E1 -5502.148,E2 -5502.148} C_VEL
LIN {X 0,Y 511.094,Z 334.977,A -85,B 0,C 180,E1 -5502.81,E2 -5502.81} C_VEL
LIN {X 0,Y 511.398,Z 323.335,A -85,B 0,C 180,E1 -5503.358,E2 -5503.358} C_VEL
LIN {X 0,Y 511.636,Z 310.831,A -85,B 0,C 180,E1 -5503.782,E2 -5503.782} C_VEL
LIN {X 0,Y 511.796,Z 298.184,A -85,B 0,C 180,E1 -5504.056,E2 -5504.056} C_VEL
LIN {X 0,Y 512.175,Z 206.462,A -85,B 0,C 180,E1 -5505.352,E2 -5505.352} C_VEL
LIN {X 0,Y 510.267,Z 194.978,A -85,B 0,C 180,E1 -5505.599,E2 -5505.599} C_VEL
LIN {X 0,Y 510.656,Z 181.028,A -85,B 0,C 180,E1 -5507.951,E2 -5507.951} C_VEL
LIN {X 0,Y 511.177,Z 161.44,A -85,B 0,C 180,E1 -5511.366,E2 -5511.366} C_VEL
LIN {X 0,Y 511.128,Z 156.662,A -85,B 0,C 180,E1 -5512.217,E2 -5512.217} C_VEL
LIN {X 0,Y 509.865,Z 150.048,A -85,B 0,C 180,E1 -5513.507,E2 -5513.507} C_VEL
LIN {X 0,Y 509.855,Z 149.965,A -85,B 0,C 180,E1 -5517.056,E2 -5517.056} C_VEL
LIN {X 0,Y 509.853,Z 149.973,A -85,B 0,C 180,E1 -5519.75,E2 -5519.75} C_VEL
LIN {X 0,Y 509.869,Z 149.973,A -85,B 0,C 180,E1 -5522.773,E2 -5522.773} C_VEL
LIN {X 0,Y 509.818,Z 149.98,A -85,B 0,C 180,E1 -5525.577,E2 -5525.577} C_VEL
LIN {X 0,Y 509.844,Z 149.966,A -85,B 0,C 180,E1 -5528.337,E2 -5528.337} C_VEL
LIN {X 0,Y 509.839,Z 149.977,A -85,B 0,C 180,E1 -5531.426,E2 -5531.426} C_VEL
LIN {X 0,Y 509.85,Z 149.974,A -85,B 0,C 180,E1 -5534.667,E2 -5534.667} C_VEL
LIN {X 0,Y 509.847,Z 149.971,A -85,B 0,C 180,E1 -5538.102,E2 -5538.102} C_VEL
LIN {X 0,Y 509.837,Z 149.976,A -85,B 0,C 180,E1 -5540.647,E2 -5540.647} C_VEL
LIN {X 0,Y 509.816,Z 149.966,A -85,B 0,C 180,E1 -5543.646,E2 -5543.646} C_VEL
LIN {X 0,Y 509.833,Z 149.974,A -85,B 0,C 180,E1 -5546.537,E2 -5546.537} C_VEL
LIN {X 0,Y 509.831,Z 149.974,A -85,B 0,C 180,E1 -5549.333,E2 -5549.333} C_VEL
LIN {X 0,Y 509.873,Z 149.968,A -85,B 0,C 180,E1 -5552.053,E2 -5552.053} C_VEL
LIN {X 0,Y 509.826,Z 149.981,A -85,B 0,C 180,E1 -5554.701,E2 -5554.701} C_VEL
LIN {X 0,Y 509.814,Z 149.976,A -85,B 0,C 180,E1 -5557.457,E2 -5557.457} C_VEL
LIN {X 0,Y 509.904,Z 149.964,A -85,B 0,C 180,E1 -5559.844,E2 -5559.844} C_VEL
LIN {X 0,Y 509.861,Z 149.971,A -85,B 0,C 180,E1 -5563.174,E2 -5563.174} C_VEL
LIN {X 0,Y 509.849,Z 149.971,A -85,B 0,C 180,E1 -5565.634,E2 -5565.634} C_VEL
LIN {X 0,Y 509.918,Z 149.965,A -85,B 0,C 180,E1 -5568.875,E2 -5568.875} C_VEL
LIN {X 0,Y 509.936,Z 149.962,A -85,B 0,C 180,E1 -5572.078,E2 -5572.078} C_VEL
LIN {X 0,Y 509.965,Z 149.961,A -85,B 0,C 180,E1 -5574.464,E2 -5574.464} C_VEL
LIN {X 0,Y 510.038,Z 149.947,A -85,B 0,C 180,E1 -5577.631,E2 -5577.631} C_VEL
LIN {X 0,Y 510.052,Z 149.947,A -85,B 0,C 180,E1 -5580.79,E2 -5580.79} C_VEL
LIN {X 0,Y 509.941,Z 149.957,A -85,B 0,C 180,E1 -5583.16,E2 -5583.16} C_VEL
LIN {X 0,Y 509.939,Z 149.967,A -85,B 0,C 180,E1 -5586.33,E2 -5586.33} C_VEL
LIN {X 0,Y 509.902,Z 149.963,A -85,B 0,C 180,E1 -5588.721,E2 -5588.721} C_VEL
LIN {X 0,Y 509.892,Z 149.968,A -85,B 0,C 180,E1 -5591.932,E2 -5591.932} C_VEL
LIN {X 0,Y 509.881,Z 149.963,A -85,B 0,C 180,E1 -5595.242,E2 -5595.242} C_VEL
LIN {X 0,Y 509.876,Z 149.971,A -85,B 0,C 180,E1 -5598.001,E2 -5598.001} C_VEL
LIN {X 0,Y 509.841,Z 149.97,A -85,B 0,C 180,E1 -5601.002,E2 -5601.002} C_VEL
LIN {X 0,Y 509.826,Z 149.973,A -85,B 0,C 180,E1 -5603.564,E2 -5603.564} C_VEL
LIN {X 0,Y 509.901,Z 149.968,A -85,B 0,C 180,E1 -5606.379,E2 -5606.379} C_VEL
LIN {X 0,Y 509.867,Z 149.969,A -85,B 0,C 180,E1 -5608.845,E2 -5608.845} C_VEL
LIN {X 0,Y 509.81,Z 149.978,A -85,B 0,C 180,E1 -5611.591,E2 -5611.591} C_VEL
LIN {X 0,Y 509.843,Z 149.962,A -85,B 0,C 180,E1 -5614.414,E2 -5614.414} C_VEL
LIN {X 0,Y 509.81,Z 149.972,A -85,B 0,C 180,E1 -5617.342,E2 -5617.342} C_VEL
LIN {X 0,Y 509.831,Z 149.976,A -85,B 0,C 180,E1 -5620.383,E2 -5620.383} C_VEL
LIN {X 0,Y 509.816,Z 149.967,A -85,B 0,C 180,E1 -5623.063,E2 -5623.063} C_VEL
LIN {X 0,Y 509.816,Z 149.979,A -85,B 0,C 180,E1 -5625.794,E2 -5625.794} C_VEL
LIN {X 0,Y 509.851,Z 149.969,A -85,B 0,C 180,E1 -5628.576,E2 -5628.576} C_VEL
LIN {X 0,Y 509.846,Z 149.975,A -85,B 0,C 180,E1 -5631.788,E2 -5631.788} C_VEL
LIN {X 0,Y 509.824,Z 149.979,A -85,B 0,C 180,E1 -5633.757,E2 -5633.757} C_VEL
LIN {X 0,Y 509.159,Z 150.056,A -85,B 0,C 180,E1 -5634.417,E2 -5634.417} C_VEL
LIN {X 0,Y 506.342,Z 150.408,A -85,B 0,C 180,E1 -5635.489,E2 -5635.489} C_VEL
LIN {X 0,Y 503.95,Z 150.709,A -85,B 0,C 180,E1 -5636.352,E2 -5636.352} C_VEL
LIN {X 0,Y 502.901,Z 150.838,A -85,B 0,C 180,E1 -5637.019,E2 -5637.019} C_VEL
LIN {X 0,Y 502.803,Z 150.849,A -85,B 0,C 180,E1 -5637.244,E2 -5637.244} C_VEL
LIN {X 0,Y 502.813,Z 150.854,A -85,B 0,C 180,E1 -5640.066,E2 -5640.066} C_VEL
LIN {X 0,Y 502.829,Z 150.849,A -85,B 0,C 180,E1 -5642.534,E2 -5642.534} C_VEL
LIN {X 0,Y 502.826,Z 150.852,A -85,B 0,C 180,E1 -5645.3,E2 -5645.3} C_VEL
LIN {X 0,Y 502.829,Z 150.946,A -85,B 0,C 180,E1 -5647.602,E2 -5647.602} C_VEL
LIN {X 0,Y 504.088,Z 158.203,A -85,B 0,C 180,E1 -5649.086,E2 -5649.086} C_VEL
LIN {X 0,Y 503.525,Z 175.641,A -85,B 0,C 180,E1 -5652.328,E2 -5652.328} C_VEL
LIN {X 0,Y 503.29,Z 186.3,A -85,B 0,C 180,E1 -5654.226,E2 -5654.226} C_VEL
LIN {X 0,Y 505.38,Z 198.17,A -85,B 0,C 180,E1 -5654.491,E2 -5654.491} C_VEL
LIN {X 0,Y 504.95,Z 293.78,A -85,B 0,C 180,E1 -5655.878,E2 -5655.878} C_VEL
LIN {X 0,Y 504.685,Z 306.934,A -85,B 0,C 180,E1 -5656.23,E2 -5656.23} C_VEL
LIN {X 0,Y 504.37,Z 319.026,A -85,B 0,C 180,E1 -5656.709,E2 -5656.709} C_VEL
LIN {X 0,Y 504.058,Z 331.148,A -85,B 0,C 180,E1 -5657.361,E2 -5657.361} C_VEL
LIN {X 0,Y 503.748,Z 342.127,A -85,B 0,C 180,E1 -5658.125,E2 -5658.125} C_VEL
LIN {X 0,Y 503.32,Z 352.622,A -85,B 0,C 180,E1 -5659.033,E2 -5659.033} C_VEL
LIN {X 0,Y 503.059,Z 361.198,A -85,B 0,C 180,E1 -5659.943,E2 -5659.943} C_VEL
LIN {X 0,Y 502.773,Z 369.1,A -85,B 0,C 180,E1 -5660.953,E2 -5660.953} C_VEL
LIN {X 0,Y 502.504,Z 376.828,A -85,B 0,C 180,E1 -5662.163,E2 -5662.163} C_VEL
LIN {X 0,Y 502.324,Z 383.918,A -85,B 0,C 180,E1 -5663.574,E2 -5663.574} C_VEL
LIN {X 0,Y 502.187,Z 388.645,A -85,B 0,C 180,E1 -5664.781,E2 -5664.781} C_VEL
LIN {X 0,Y 502.186,Z 392.265,A -85,B 0,C 180,E1 -5665.988,E2 -5665.988} C_VEL
LIN {X 0,Y 502.14,Z 394.137,A -85,B 0,C 180,E1 -5666.791,E2 -5666.791} C_VEL
LIN {X 0,Y 502.096,Z 395.549,A -85,B 0,C 180,E1 -5667.594,E2 -5667.594} C_VEL
LIN {X 0,Y 501.991,Z 397.172,A -85,B 0,C 180,E1 -5669.198,E2 -5669.198} C_VEL
LIN {X 0,Y 501.981,Z 397.41,A -85,B 0,C 180,E1 -5670,E2 -5670} C_VEL
LIN {X 0,Y 501.991,Z 397.225,A -85,B 0,C 180,E1 -5670.803,E2 -5670.803} C_VEL
LIN {X 0,Y 502.096,Z 395.671,A -85,B 0,C 180,E1 -5672.407,E2 -5672.407} C_VEL
LIN {X 0,Y 502.141,Z 394.311,A -85,B 0,C 180,E1 -5673.21,E2 -5673.21} C_VEL
LIN {X 0,Y 502.148,Z 391.437,A -85,B 0,C 180,E1 -5674.415,E2 -5674.415} C_VEL
LIN {X 0,Y 502.29,Z 387.54,A -85,B 0,C 180,E1 -5675.621,E2 -5675.621} C_VEL
LIN {X 0,Y 502.353,Z 382.515,A -85,B 0,C 180,E1 -5676.829,E2 -5676.829} C_VEL
LIN {X 0,Y 502.519,Z 376.189,A -85,B 0,C 180,E1 -5678.04,E2 -5678.04} C_VEL
LIN {X 0,Y 502.772,Z 368.271,A -85,B 0,C 180,E1 -5679.251,E2 -5679.251} C_VEL
LIN {X 0,Y 503.042,Z 360.201,A -85,B 0,C 180,E1 -5680.261,E2 -5680.261} C_VEL
LIN {X 0,Y 503.423,Z 350.356,A -85,B 0,C 180,E1 -5681.271,E2 -5681.271} C_VEL
LIN {X 0,Y 503.79,Z 339.317,A -85,B 0,C 180,E1 -5682.179,E2 -5682.179} C_VEL
LIN {X 0,Y 504.133,Z 328.454,A -85,B 0,C 180,E1 -5682.888,E2 -5682.888} C_VEL
LIN {X 0,Y 504.455,Z 316.488,A -85,B 0,C 180,E1 -5683.495,E2 -5683.495} C_VEL
LIN {X 0,Y 504.762,Z 303.395,A -85,B 0,C 180,E1 -5683.974,E2 -5683.974} C_VEL
LIN {X 0,Y 504.994,Z 290.26,A -85,B 0,C 180,E1 -5684.276,E2 -5684.276} C_VEL
LIN {X 0,Y 505.273,Z 197.636,A -85,B 0,C 180,E1 -5685.61,E2 -5685.61} C_VEL
LIN {X 0,Y 503.321,Z 186.42,A -85,B 0,C 180,E1 -5685.856,E2 -5685.856} C_VEL
LIN {X 0,Y 503.308,Z 184.092,A -85,B 0,C 180,E1 -5686.217,E2 -5686.217} C_VEL
LIN {X 0,Y 503.766,Z 167.062,A -85,B 0,C 180,E1 -5689.35,E2 -5689.35} C_VEL
LIN {X 0,Y 503.981,Z 156.892,A -85,B 0,C 180,E1 -5691.258,E2 -5691.258} C_VEL
LIN {X 0,Y 502.812,Z 150.98,A -85,B 0,C 180,E1 -5692.476,E2 -5692.476} C_VEL
LIN {X 0,Y 502.842,Z 150.848,A -85,B 0,C 180,E1 -5695.675,E2 -5695.675} C_VEL
LIN {X 0,Y 502.84,Z 150.849,A -85,B 0,C 180,E1 -5698.372,E2 -5698.372} C_VEL
LIN {X 0,Y 502.793,Z 150.847,A -85,B 0,C 180,E1 -5701.498,E2 -5701.498} C_VEL
LIN {X 0,Y 502.804,Z 150.849,A -85,B 0,C 180,E1 -5704.444,E2 -5704.444} C_VEL
LIN {X 0,Y 502.78,Z 150.853,A -85,B 0,C 180,E1 -5707.178,E2 -5707.178} C_VEL
LIN {X 0,Y 502.786,Z 150.849,A -85,B 0,C 180,E1 -5710.015,E2 -5710.015} C_VEL
LIN {X 0,Y 502.801,Z 150.855,A -85,B 0,C 180,E1 -5712.199,E2 -5712.199} C_VEL
LIN {X 0,Y 502.783,Z 150.85,A -85,B 0,C 180,E1 -5715.469,E2 -5715.469} C_VEL
LIN {X 0,Y 502.818,Z 150.846,A -85,B 0,C 180,E1 -5718.934,E2 -5718.934} C_VEL
LIN {X 0,Y 502.79,Z 150.855,A -85,B 0,C 180,E1 -5722.045,E2 -5722.045} C_VEL
LIN {X 0,Y 502.801,Z 150.833,A -85,B 0,C 180,E1 -5725.034,E2 -5725.034} C_VEL
LIN {X 0,Y 502.778,Z 150.855,A -85,B 0,C 180,E1 -5727.915,E2 -5727.915} C_VEL
LIN {X 0,Y 502.819,Z 150.847,A -85,B 0,C 180,E1 -5730.712,E2 -5730.712} C_VEL
LIN {X 0,Y 502.857,Z 150.842,A -85,B 0,C 180,E1 -5733.439,E2 -5733.439} C_VEL
LIN {X 0,Y 502.768,Z 150.857,A -85,B 0,C 180,E1 -5736.085,E2 -5736.085} C_VEL
LIN {X 0,Y 502.776,Z 150.849,A -85,B 0,C 180,E1 -5738.688,E2 -5738.688} C_VEL
LIN {X 0,Y 502.822,Z 150.849,A -85,B 0,C 180,E1 -5741.248,E2 -5741.248} C_VEL
LIN {X 0,Y 502.815,Z 150.85,A -85,B 0,C 180,E1 -5743.767,E2 -5743.767} C_VEL
LIN {X 0,Y 502.823,Z 150.848,A -85,B 0,C 180,E1 -5746.254,E2 -5746.254} C_VEL
LIN {X 0,Y 502.869,Z 150.84,A -85,B 0,C 180,E1 -5748.717,E2 -5748.717} C_VEL
LIN {X 0,Y 502.894,Z 150.84,A -85,B 0,C 180,E1 -5751.966,E2 -5751.966} C_VEL
LIN {X 0,Y 502.923,Z 150.834,A -85,B 0,C 180,E1 -5754.386,E2 -5754.386} C_VEL
LIN {X 0,Y 503.014,Z 150.824,A -85,B 0,C 180,E1 -5757.598,E2 -5757.598} C_VEL
LIN {X 0,Y 503.015,Z 150.825,A -85,B 0,C 180,E1 -5760,E2 -5760} C_VEL
LIN {X 0,Y 503.013,Z 150.822,A -85,B 0,C 180,E1 -5762.402,E2 -5762.402} C_VEL
LIN {X 0,Y 502.923,Z 150.839,A -85,B 0,C 180,E1 -5765.614,E2 -5765.614} C_VEL
LIN {X 0,Y 502.872,Z 150.842,A -85,B 0,C 180,E1 -5768.034,E2 -5768.034} C_VEL
LIN {X 0,Y 502.868,Z 150.843,A -85,B 0,C 180,E1 -5771.283,E2 -5771.283} C_VEL
LIN {X 0,Y 502.836,Z 150.845,A -85,B 0,C 180,E1 -5774.571,E2 -5774.571} C_VEL
LIN {X 0,Y 502.815,Z 150.844,A -85,B 0,C 180,E1 -5777.909,E2 -5777.909} C_VEL
LIN {X 0,Y 502.822,Z 150.847,A -85,B 0,C 180,E1 -5780.536,E2 -5780.536} C_VEL
LIN {X 0,Y 502.781,Z 150.857,A -85,B 0,C 180,E1 -5783.041,E2 -5783.041} C_VEL
LIN {X 0,Y 502.813,Z 150.85,A -85,B 0,C 180,E1 -5785.677,E2 -5785.677} C_VEL
LIN {X 0,Y 502.831,Z 150.845,A -85,B 0,C 180,E1 -5788.373,E2 -5788.373} C_VEL
LIN {X 0,Y 502.786,Z 150.855,A -85,B 0,C 180,E1 -5791.499,E2 -5791.499} C_VEL
LIN {X 0,Y 502.784,Z 150.849,A -85,B 0,C 180,E1 -5793.996,E2 -5793.996} C_VEL
LIN {X 0,Y 502.772,Z 150.848,A -85,B 0,C 180,E1 -5797.178,E2 -5797.178} C_VEL
LIN {X 0,Y 502.783,Z 150.851,A -85,B 0,C 180,E1 -5800.016,E2 -5800.016} C_VEL
LIN {X 0,Y 502.8,Z 150.849,A -85,B 0,C 180,E1 -5802.2,E2 -5802.2} C_VEL
LIN {X 0,Y 502.782,Z 150.853,A -85,B 0,C 180,E1 -5805.471,E2 -5805.471} C_VEL
LIN {X 0,Y 502.792,Z 150.85,A -85,B 0,C 180,E1 -5807.861,E2 -5807.861} C_VEL
LIN {X 0,Y 502.794,Z 150.848,A -85,B 0,C 180,E1 -5811.024,E2 -5811.024} C_VEL
LIN {X 0,Y 502.77,Z 150.856,A -85,B 0,C 180,E1 -5814.17,E2 -5814.17} C_VEL
LIN {X 0,Y 502.832,Z 150.852,A -85,B 0,C 180,E1 -5816.994,E2 -5816.994} C_VEL
LIN {X 0,Y 502.814,Z 150.848,A -85,B 0,C 180,E1 -5820.066,E2 -5820.066} C_VEL
LIN {X 0,Y 502.844,Z 150.84,A -85,B 0,C 180,E1 -5823.444,E2 -5823.444} C_VEL
LIN {X 0,Y 502.823,Z 150.909,A -85,B 0,C 180,E1 -5826.307,E2 -5826.307} C_VEL
LIN {X 0,Y 503.546,Z 154.762,A -85,B 0,C 180,E1 -5827.097,E2 -5827.097} C_VEL
LIN {X 0,Y 504.292,Z 158.991,A -85,B 0,C 180,E1 -5827.897,E2 -5827.897} C_VEL
LIN {X 0,Y 503.853,Z 173.305,A -85,B 0,C 180,E1 -5830.442,E2 -5830.442} C_VEL
LIN {X 0,Y 503.427,Z 187.61,A -85,B 0,C 180,E1 -5832.952,E2 -5832.952} C_VEL
LIN {X 0,Y 503.274,Z 194.86,A -85,B 0,C 180,E1 -5834.174,E2 -5834.174} C_VEL
LIN {X 0,Y 505.361,Z 207.623,A -85,B 0,C 180,E1 -5834.453,E2 -5834.453} C_VEL
LIN {X 0,Y 504.924,Z 302.43,A -85,B 0,C 180,E1 -5835.825,E2 -5835.825} C_VEL
LIN {X 0,Y 504.584,Z 315.703,A -85,B 0,C 180,E1 -5836.175,E2 -5836.175} C_VEL
LIN {X 0,Y 504.302,Z 327.86,A -85,B 0,C 180,E1 -5836.655,E2 -5836.655} C_VEL
LIN {X 0,Y 504.008,Z 339.623,A -85,B 0,C 180,E1 -5837.281,E2 -5837.281} C_VEL
LIN {X 0,Y 503.691,Z 350.41,A -85,B 0,C 180,E1 -5838.021,E2 -5838.021} C_VEL
LIN {X 0,Y 503.316,Z 361.056,A -85,B 0,C 180,E1 -5838.931,E2 -5838.931} C_VEL
LIN {X 0,Y 502.957,Z 370.645,A -85,B 0,C 180,E1 -5839.941,E2 -5839.941} C_VEL
LIN {X 0,Y 502.669,Z 378.504,A -85,B 0,C 180,E1 -5840.95,E2 -5840.95} C_VEL
LIN {X 0,Y 502.446,Z 386.176,A -85,B 0,C 180,E1 -5842.161,E2 -5842.161} C_VEL
LIN {X 0,Y 502.235,Z 393.247,A -85,B 0,C 180,E1 -5843.572,E2 -5843.572} C_VEL
LIN {X 0,Y 502.18,Z 397.95,A -85,B 0,C 180,E1 -5844.781,E2 -5844.781} C_VEL
LIN {X 0,Y 502.14,Z 401.542,A -85,B 0,C 180,E1 -5845.987,E2 -5845.987} C_VEL
LIN {X 0,Y 502.12,Z 403.395,A -85,B 0,C 180,E1 -5846.79,E2 -5846.79} C_VEL
LIN {X 0,Y 502.036,Z 405.775,A -85,B 0,C 180,E1 -5848.395,E2 -5848.395} C_VEL
LIN {X 0,Y 501.98,Z 406.595,A -85,B 0,C 180,E1 -5850,E2 -5850} C_VEL
LIN {X 0,Y 502.035,Z 405.777,A -85,B 0,C 180,E1 -5851.604,E2 -5851.604} C_VEL
LIN {X 0,Y 502.12,Z 403.4,A -85,B 0,C 180,E1 -5853.209,E2 -5853.209} C_VEL
LIN {X 0,Y 502.103,Z 400.479,A -85,B 0,C 180,E1 -5854.415,E2 -5854.415} C_VEL
LIN {X 0,Y 502.23,Z 396.525,A -85,B 0,C 180,E1 -5855.621,E2 -5855.621} C_VEL
LIN {X 0,Y 502.332,Z 390.543,A -85,B 0,C 180,E1 -5857.011,E2 -5857.011} C_VEL
LIN {X 0,Y 502.523,Z 383.791,A -85,B 0,C 180,E1 -5858.241,E2 -5858.241} C_VEL
LIN {X 0,Y 502.759,Z 375.536,A -85,B 0,C 180,E1 -5859.453,E2 -5859.453} C_VEL
LIN {X 0,Y 503.049,Z 367.074,A -85,B 0,C 180,E1 -5860.464,E2 -5860.464} C_VEL
LIN {X 0,Y 503.449,Z 356.614,A -85,B 0,C 180,E1 -5861.474,E2 -5861.474} C_VEL
LIN {X 0,Y 503.772,Z 345.766,A -85,B 0,C 180,E1 -5862.318,E2 -5862.318} C_VEL
LIN {X 0,Y 504.15,Z 334.911,A -85,B 0,C 180,E1 -5862.99,E2 -5862.99} C_VEL
LIN {X 0,Y 504.476,Z 323.268,A -85,B 0,C 180,E1 -5863.545,E2 -5863.545} C_VEL
LIN {X 0,Y 504.724,Z 310.763,A -85,B 0,C 180,E1 -5863.975,E2 -5863.975} C_VEL
LIN {X 0,Y 504.938,Z 298.114,A -85,B 0,C 180,E1 -5864.251,E2 -5864.251} C_VEL
LIN {X 0,Y 505.261,Z 206.753,A -85,B 0,C 180,E1 -5865.562,E2 -5865.562} C_VEL
LIN {X 0,Y 503.274,Z 194.876,A -85,B 0,C 180,E1 -5865.824,E2 -5865.824} C_VEL
LIN {X 0,Y 503.709,Z 179.762,A -85,B 0,C 180,E1 -5868.419,E2 -5868.419} C_VEL
LIN {X 0,Y 504.272,Z 161.375,A -85,B 0,C 180,E1 -5871.673,E2 -5871.673} C_VEL
LIN {X 0,Y 504.139,Z 157.859,A -85,B 0,C 180,E1 -5872.313,E2 -5872.313} C_VEL
LIN {X 0,Y 502.858,Z 151.233,A -85,B 0,C 180,E1 -5873.581,E2 -5873.581} C_VEL
LIN {X 0,Y 502.781,Z 150.847,A -85,B 0,C 180,E1 -5873.913,E2 -5873.913} C_VEL
LIN {X 0,Y 502.833,Z 150.841,A -85,B 0,C 180,E1 -5876.567,E2 -5876.567} C_VEL
LIN {X 0,Y 502.811,Z 150.849,A -85,B 0,C 180,E1 -5879.934,E2 -5879.934} C_VEL
LIN {X 0,Y 502.828,Z 150.852,A -85,B 0,C 180,E1 -5883.03,E2 -5883.03} C_VEL
LIN {X 0,Y 502.763,Z 150.856,A -85,B 0,C 180,E1 -5885.951,E2 -5885.951} C_VEL
LIN {X 0,Y 502.795,Z 150.848,A -85,B 0,C 180,E1 -5888.975,E2 -5888.975} C_VEL
LIN {X 0,Y 502.797,Z 150.85,A -85,B 0,C 180,E1 -5892.198,E2 -5892.198} C_VEL
LIN {X 0,Y 502.793,Z 150.852,A -85,B 0,C 180,E1 -5895.467,E2 -5895.467} C_VEL
LIN {X 0,Y 502.811,Z 150.855,A -85,B 0,C 180,E1 -5898.933,E2 -5898.933} C_VEL
LIN {X 0,Y 502.783,Z 150.845,A -85,B 0,C 180,E1 -5902.045,E2 -5902.045} C_VEL
LIN {X 0,Y 502.788,Z 150.85,A -85,B 0,C 180,E1 -5905.033,E2 -5905.033} C_VEL
LIN {X 0,Y 502.771,Z 150.853,A -85,B 0,C 180,E1 -5907.914,E2 -5907.914} C_VEL
LIN {X 0,Y 502.811,Z 150.851,A -85,B 0,C 180,E1 -5910.711,E2 -5910.711} C_VEL
LIN {X 0,Y 502.851,Z 150.845,A -85,B 0,C 180,E1 -5913.439,E2 -5913.439} C_VEL
LIN {X 0,Y 502.762,Z 150.85,A -85,B 0,C 180,E1 -5916.085,E2 -5916.085} C_VEL
LIN {X 0,Y 502.771,Z 150.86,A -85,B 0,C 180,E1 -5918.688,E2 -5918.688} C_VEL
LIN {X 0,Y 502.814,Z 150.845,A -85,B 0,C 180,E1 -5921.248,E2 -5921.248} C_VEL
LIN {X 0,Y 502.836,Z 150.851,A -85,B 0,C 180,E1 -5924.6,E2 -5924.6} C_VEL
LIN {X 0,Y 502.886,Z 150.836,A -85,B 0,C 180,E1 -5928.026,E2 -5928.026} C_VEL
LIN {X 0,Y 502.858,Z 150.844,A -85,B 0,C 180,E1 -5931.156,E2 -5931.156} C_VEL
LIN {X 0,Y 502.892,Z 150.836,A -85,B 0,C 180,E1 -5933.581,E2 -5933.581} C_VEL
LIN {X 0,Y 502.886,Z 150.843,A -85,B 0,C 180,E1 -5936.795,E2 -5936.795} C_VEL
LIN {X 0,Y 503.021,Z 150.823,A -85,B 0,C 180,E1 -5939.199,E2 -5939.199} C_VEL
LIN {X 0,Y 502.885,Z 150.835,A -85,B 0,C 180,E1 -5941.602,E2 -5941.602} C_VEL
LIN {X 0,Y 502.884,Z 150.836,A -85,B 0,C 180,E1 -5943.205,E2 -5943.205} C_VEL
LIN {X 0,Y 502.892,Z 150.846,A -85,B 0,C 180,E1 -5946.419,E2 -5946.419} C_VEL
LIN {X 0,Y 502.861,Z 150.838,A -85,B 0,C 180,E1 -5948.844,E2 -5948.844} C_VEL
LIN {X 0,Y 502.833,Z 150.849,A -85,B 0,C 180,E1 -5952.102,E2 -5952.102} C_VEL
LIN {X 0,Y 502.836,Z 150.84,A -85,B 0,C 180,E1 -5955.4,E2 -5955.4} C_VEL
LIN {X 0,Y 502.834,Z 150.85,A -85,B 0,C 180,E1 -5958.123,E2 -5958.123} C_VEL
LIN {X 0,Y 502.817,Z 150.849,A -85,B 0,C 180,E1 -5960.537,E2 -5960.537} C_VEL
LIN {X 0,Y 502.789,Z 150.849,A -85,B 0,C 180,E1 -5963.041,E2 -5963.041} C_VEL
LIN {X 0,Y 502.829,Z 150.848,A -85,B 0,C 180,E1 -5965.676,E2 -5965.676} C_VEL
LIN {X 0,Y 502.83,Z 150.85,A -85,B 0,C 180,E1 -5968.373,E2 -5968.373} C_VEL
LIN {X 0,Y 502.783,Z 150.853,A -85,B 0,C 180,E1 -5971.5,E2 -5971.5} C_VEL
LIN {X 0,Y 502.795,Z 150.839,A -85,B 0,C 180,E1 -5974.445,E2 -5974.445} C_VEL
LIN {X 0,Y 502.772,Z 150.848,A -85,B 0,C 180,E1 -5977.179,E2 -5977.179} C_VEL
LIN {X 0,Y 502.78,Z 150.86,A -85,B 0,C 180,E1 -5980.016,E2 -5980.016} C_VEL
LIN {X 0,Y 502.796,Z 150.847,A -85,B 0,C 180,E1 -5982.2,E2 -5982.2} C_VEL
LIN {X 0,Y 502.779,Z 150.851,A -85,B 0,C 180,E1 -5985.471,E2 -5985.471} C_VEL
LIN {X 0,Y 502.815,Z 150.844,A -85,B 0,C 180,E1 -5988.935,E2 -5988.935} C_VEL
LIN {X 0,Y 502.789,Z 150.858,A -85,B 0,C 180,E1 -5992.047,E2 -5992.047} C_VEL
LIN {X 0,Y 502.802,Z 150.846,A -85,B 0,C 180,E1 -5995.036,E2 -5995.036} C_VEL
LIN {X 0,Y 502.803,Z 150.849,A -85,B 0,C 180,E1 -5997.244,E2 -5997.244} C_VEL
LIN {X 0,Y 502.103,Z 150.941,A -85,B 0,C 180,E1 -5997.913,E2 -5997.913} C_VEL
LIN {X 0,Y 499.238,Z 151.294,A -85,B 0,C 180,E1 -5998.999,E2 -5998.999} C_VEL
LIN {X 0,Y 496.844,Z 151.599,A -85,B 0,C 180,E1 -5999.874,E2 -5999.874} C_VEL
LIN {X 0,Y 495.828,Z 151.72,A -85,B 0,C 180,E1 -6000.549,E2 -6000.549} C_VEL
LIN {X 0,Y 495.751,Z 151.729,A -85,B 0,C 180,E1 -6000.778,E2 -6000.778} C_VEL
LIN {X 0,Y 495.79,Z 151.728,A -85,B 0,C 180,E1 -6003.933,E2 -6003.933} C_VEL
LIN {X 0,Y 495.77,Z 151.759,A -85,B 0,C 180,E1 -6007.398,E2 -6007.398} C_VEL
LIN {X 0,Y 496.456,Z 155.306,A -85,B 0,C 180,E1 -6008.186,E2 -6008.186} C_VEL
LIN {X 0,Y 497.085,Z 159.016,A -85,B 0,C 180,E1 -6008.93,E2 -6008.93} C_VEL
LIN {X 0,Y 496.589,Z 175.686,A -85,B 0,C 180,E1 -6012.073,E2 -6012.073} C_VEL
LIN {X 0,Y 496.296,Z 186.238,A -85,B 0,C 180,E1 -6013.987,E2 -6013.987} C_VEL
LIN {X 0,Y 497.434,Z 192.621,A -85,B 0,C 180,E1 -6014.154,E2 -6014.154} C_VEL
LIN {X 0,Y 498.525,Z 199.518,A -85,B 0,C 180,E1 -6014.291,E2 -6014.291} C_VEL
LIN {X 0,Y 498.091,Z 293.866,A -85,B 0,C 180,E1 -6015.679,E2 -6015.679} C_VEL
LIN {X 0,Y 497.81,Z 307.013,A -85,B 0,C 180,E1 -6016.036,E2 -6016.036} C_VEL
LIN {X 0,Y 497.447,Z 319.102,A -85,B 0,C 180,E1 -6016.52,E2 -6016.52} C_VEL
LIN {X 0,Y 497.11,Z 331.301,A -85,B 0,C 180,E1 -6017.186,E2 -6017.186} C_VEL
LIN {X 0,Y 496.806,Z 342.199,A -85,B 0,C 180,E1 -6017.957,E2 -6017.957} C_VEL
LIN {X 0,Y 496.343,Z 352.693,A -85,B 0,C 180,E1 -6018.877,E2 -6018.877} C_VEL
LIN {X 0,Y 496.056,Z 361.268,A -85,B 0,C 180,E1 -6019.8,E2 -6019.8} C_VEL
LIN {X 0,Y 495.726,Z 369.169,A -85,B 0,C 180,E1 -6020.823,E2 -6020.823} C_VEL
LIN {X 0,Y 495.453,Z 376.896,A -85,B 0,C 180,E1 -6022.051,E2 -6022.051} C_VEL
LIN {X 0,Y 495.252,Z 383.986,A -85,B 0,C 180,E1 -6023.482,E2 -6023.482} C_VEL
LIN {X 0,Y 495.129,Z 388.712,A -85,B 0,C 180,E1 -6024.707,E2 -6024.707} C_VEL
LIN {X 0,Y 495.085,Z 392.332,A -85,B 0,C 180,E1 -6025.93,E2 -6025.93} C_VEL
LIN {X 0,Y 495.062,Z 394.203,A -85,B 0,C 180,E1 -6026.745,E2 -6026.745} C_VEL
LIN {X 0,Y 495.003,Z 395.615,A -85,B 0,C 180,E1 -6027.559,E2 -6027.559} C_VEL
LIN {X 0,Y 494.911,Z 397.237,A -85,B 0,C 180,E1 -6029.187,E2 -6029.187} C_VEL
LIN {X 0,Y 494.899,Z 397.475,A -85,B 0,C 180,E1 -6030,E2 -6030} C_VEL
LIN {X 0,Y 494.911,Z 397.29,A -85,B 0,C 180,E1 -6030.814,E2 -6030.814} C_VEL
LIN {X 0,Y 495.003,Z 395.735,A -85,B 0,C 180,E1 -6032.441,E2 -6032.441} C_VEL
LIN {X 0,Y 495.062,Z 394.375,A -85,B 0,C 180,E1 -6033.256,E2 -6033.256} C_VEL
LIN {X 0,Y 495.046,Z 391.501,A -85,B 0,C 180,E1 -6034.479,E2 -6034.479} C_VEL
LIN {X 0,Y 495.208,Z 387.603,A -85,B 0,C 180,E1 -6035.702,E2 -6035.702} C_VEL
LIN {X 0,Y 495.287,Z 382.577,A -85,B 0,C 180,E1 -6036.927,E2 -6036.927} C_VEL
LIN {X 0,Y 495.481,Z 376.25,A -85,B 0,C 180,E1 -6038.155,E2 -6038.155} C_VEL
LIN {X 0,Y 495.752,Z 368.332,A -85,B 0,C 180,E1 -6039.383,E2 -6039.383} C_VEL
LIN {X 0,Y 496.043,Z 360.262,A -85,B 0,C 180,E1 -6040.407,E2 -6040.407} C_VEL
LIN {X 0,Y 496.468,Z 350.416,A -85,B 0,C 180,E1 -6041.431,E2 -6041.431} C_VEL
LIN {X 0,Y 496.818,Z 340.734,A -85,B 0,C 180,E1 -6042.251,E2 -6042.251} C_VEL
LIN {X 0,Y 497.137,Z 330.112,A -85,B 0,C 180,E1 -6042.979,E2 -6042.979} C_VEL
LIN {X 0,Y 497.54,Z 317.671,A -85,B 0,C 180,E1 -6043.634,E2 -6043.634} C_VEL
LIN {X 0,Y 497.87,Z 304.307,A -85,B 0,C 180,E1 -6044.146,E2 -6044.146} C_VEL
LIN {X 0,Y 498.12,Z 291.801,A -85,B 0,C 180,E1 -6044.451,E2 -6044.451} C_VEL
LIN {X 0,Y 498.514,Z 198.897,A -85,B 0,C 180,E1 -6045.809,E2 -6045.809} C_VEL
LIN {X 0,Y 496.296,Z 186.361,A -85,B 0,C 180,E1 -6046.093,E2 -6046.093} C_VEL
LIN {X 0,Y 496.456,Z 179.582,A -85,B 0,C 180,E1 -6047.294,E2 -6047.294} C_VEL
LIN {X 0,Y 497.032,Z 162.56,A -85,B 0,C 180,E1 -6050.485,E2 -6050.485} C_VEL
LIN {X 0,Y 497.042,Z 158.524,A -85,B 0,C 180,E1 -6051.258,E2 -6051.258} C_VEL
LIN {X 0,Y 495.769,Z 151.807,A -85,B 0,C 180,E1 -6052.669,E2 -6052.669} C_VEL
LIN {X 0,Y 495.793,Z 151.729,A -85,B 0,C 180,E1 -6056.067,E2 -6056.067} C_VEL
LIN {X 0,Y 495.772,Z 151.729,A -85,B 0,C 180,E1 -6058.814,E2 -6058.814} C_VEL
LIN {X 0,Y 495.756,Z 151.725,A -85,B 0,C 180,E1 -6061.725,E2 -6061.725} C_VEL
LIN {X 0,Y 495.774,Z 151.723,A -85,B 0,C 180,E1 -6064.694,E2 -6064.694} C_VEL
LIN {X 0,Y 495.73,Z 151.732,A -85,B 0,C 180,E1 -6067.561,E2 -6067.561} C_VEL
LIN {X 0,Y 495.765,Z 151.724,A -85,B 0,C 180,E1 -6070.699,E2 -6070.699} C_VEL
LIN {X 0,Y 495.726,Z 151.738,A -85,B 0,C 180,E1 -6074.001,E2 -6074.001} C_VEL
LIN {X 0,Y 495.721,Z 151.721,A -85,B 0,C 180,E1 -6077.116,E2 -6077.116} C_VEL
LIN {X 0,Y 495.756,Z 151.733,A -85,B 0,C 180,E1 -6079.952,E2 -6079.952} C_VEL
LIN {X 0,Y 495.726,Z 151.728,A -85,B 0,C 180,E1 -6082.552,E2 -6082.552} C_VEL
LIN {X 0,Y 495.777,Z 151.709,A -85,B 0,C 180,E1 -6085.456,E2 -6085.456} C_VEL
LIN {X 0,Y 495.75,Z 151.731,A -85,B 0,C 180,E1 -6088.363,E2 -6088.363} C_VEL
LIN {X 0,Y 495.783,Z 151.726,A -85,B 0,C 180,E1 -6091.506,E2 -6091.506} C_VEL
LIN {X 0,Y 495.775,Z 151.731,A -85,B 0,C 180,E1 -6093.931,E2 -6093.931} C_VEL
LIN {X 0,Y 495.752,Z 151.726,A -85,B 0,C 180,E1 -6097.139,E2 -6097.139} C_VEL
LIN {X 0,Y 495.764,Z 151.73,A -85,B 0,C 180,E1 -6100.109,E2 -6100.109} C_VEL
LIN {X 0,Y 495.775,Z 151.723,A -85,B 0,C 180,E1 -6102.681,E2 -6102.681} C_VEL
LIN {X 0,Y 495.783,Z 151.72,A -85,B 0,C 180,E1 -6105.217,E2 -6105.217} C_VEL
LIN {X 0,Y 495.844,Z 151.715,A -85,B 0,C 180,E1 -6108.555,E2 -6108.555} C_VEL
LIN {X 0,Y 495.865,Z 151.717,A -85,B 0,C 180,E1 -6111.852,E2 -6111.852} C_VEL
LIN {X 0,Y 495.88,Z 151.712,A -85,B 0,C 180,E1 -6114.306,E2 -6114.306} C_VEL
LIN {X 0,Y 495.983,Z 151.699,A -85,B 0,C 180,E1 -6117.564,E2 -6117.564} C_VEL
LIN {X 0,Y 495.987,Z 151.701,A -85,B 0,C 180,E1 -6120,E2 -6120} C_VEL
LIN {X 0,Y 495.982,Z 151.698,A -85,B 0,C 180,E1 -6122.436,E2 -6122.436} C_VEL
LIN {X 0,Y 495.879,Z 151.715,A -85,B 0,C 180,E1 -6125.694,E2 -6125.694} C_VEL
LIN {X 0,Y 495.828,Z 151.718,A -85,B 0,C 180,E1 -6128.149,E2 -6128.149} C_VEL
LIN {X 0,Y 495.843,Z 151.717,A -85,B 0,C 180,E1 -6131.445,E2 -6131.445} C_VEL
LIN {X 0,Y 495.782,Z 151.726,A -85,B 0,C 180,E1 -6134.783,E2 -6134.783} C_VEL
LIN {X 0,Y 495.756,Z 151.729,A -85,B 0,C 180,E1 -6137.32,E2 -6137.32} C_VEL
LIN {X 0,Y 495.762,Z 151.727,A -85,B 0,C 180,E1 -6139.891,E2 -6139.891} C_VEL
LIN {X 0,Y 495.752,Z 151.73,A -85,B 0,C 180,E1 -6142.861,E2 -6142.861} C_VEL
LIN {X 0,Y 495.773,Z 151.725,A -85,B 0,C 180,E1 -6146.069,E2 -6146.069} C_VEL
LIN {X 0,Y 495.763,Z 151.729,A -85,B 0,C 180,E1 -6148.815,E2 -6148.815} C_VEL
LIN {X 0,Y 495.748,Z 151.73,A -85,B 0,C 180,E1 -6151.725,E2 -6151.725} C_VEL
LIN {X 0,Y 495.757,Z 151.727,A -85,B 0,C 180,E1 -6154.693,E2 -6154.693} C_VEL
LIN {X 0,Y 495.724,Z 151.726,A -85,B 0,C 180,E1 -6157.562,E2 -6157.562} C_VEL
LIN {X 0,Y 495.754,Z 151.727,A -85,B 0,C 180,E1 -6160.047,E2 -6160.047} C_VEL
LIN {X 0,Y 495.711,Z 151.736,A -85,B 0,C 180,E1 -6162.885,E2 -6162.885} C_VEL
LIN {X 0,Y 495.721,Z 151.731,A -85,B 0,C 180,E1 -6165.998,E2 -6165.998} C_VEL
LIN {X 0,Y 495.733,Z 151.732,A -85,B 0,C 180,E1 -6169.297,E2 -6169.297} C_VEL
LIN {X 0,Y 495.746,Z 151.723,A -85,B 0,C 180,E1 -6171.409,E2 -6171.409} C_VEL
LIN {X 0,Y 495.744,Z 151.734,A -85,B 0,C 180,E1 -6174.463,E2 -6174.463} C_VEL
LIN {X 0,Y 495.767,Z 151.729,A -85,B 0,C 180,E1 -6177.406,E2 -6177.406} C_VEL
LIN {X 0,Y 495.762,Z 151.728,A -85,B 0,C 180,E1 -6180.254,E2 -6180.254} C_VEL
LIN {X 0,Y 495.775,Z 151.718,A -85,B 0,C 180,E1 -6183.263,E2 -6183.263} C_VEL
LIN {X 0,Y 495.771,Z 151.892,A -85,B 0,C 180,E1 -6186.171,E2 -6186.171} C_VEL
LIN {X 0,Y 497.329,Z 160.122,A -85,B 0,C 180,E1 -6187.789,E2 -6187.789} C_VEL
LIN {X 0,Y 496.969,Z 172.05,A -85,B 0,C 180,E1 -6189.944,E2 -6189.944} C_VEL
LIN {X 0,Y 496.492,Z 187.547,A -85,B 0,C 180,E1 -6192.707,E2 -6192.707} C_VEL
LIN {X 0,Y 496.304,Z 194.595,A -85,B 0,C 180,E1 -6193.928,E2 -6193.928} C_VEL
LIN {X 0,Y 496.873,Z 198.498,A -85,B 0,C 180,E1 -6194.048,E2 -6194.048} C_VEL
LIN {X 0,Y 498.581,Z 208.918,A -85,B 0,C 180,E1 -6194.256,E2 -6194.256} C_VEL
LIN {X 0,Y 498.048,Z 302.372,A -85,B 0,C 180,E1 -6195.625,E2 -6195.625} C_VEL
LIN {X 0,Y 497.715,Z 315.643,A -85,B 0,C 180,E1 -6195.98,E2 -6195.98} C_VEL
LIN {X 0,Y 497.41,Z 327.798,A -85,B 0,C 180,E1 -6196.466,E2 -6196.466} C_VEL
LIN {X 0,Y 497.053,Z 339.838,A -85,B 0,C 180,E1 -6197.118,E2 -6197.118} C_VEL
LIN {X 0,Y 496.724,Z 350.347,A -85,B 0,C 180,E1 -6197.851,E2 -6197.851} C_VEL
LIN {X 0,Y 496.343,Z 360.992,A -85,B 0,C 180,E1 -6198.773,E2 -6198.773} C_VEL
LIN {X 0,Y 495.929,Z 370.581,A -85,B 0,C 180,E1 -6199.797,E2 -6199.797} C_VEL
LIN {X 0,Y 495.644,Z 378.439,A -85,B 0,C 180,E1 -6200.821,E2 -6200.821} C_VEL
LIN {X 0,Y 495.378,Z 386.112,A -85,B 0,C 180,E1 -6202.049,E2 -6202.049} C_VEL
LIN {X 0,Y 495.164,Z 393.182,A -85,B 0,C 180,E1 -6203.48,E2 -6203.48} C_VEL
LIN {X 0,Y 495.114,Z 397.885,A -85,B 0,C 180,E1 -6204.706,E2 -6204.706} C_VEL
LIN {X 0,Y 495.034,Z 401.477,A -85,B 0,C 180,E1 -6205.929,E2 -6205.929} C_VEL
LIN {X 0,Y 495.042,Z 403.33,A -85,B 0,C 180,E1 -6206.744,E2 -6206.744} C_VEL
LIN {X 0,Y 494.961,Z 405.71,A -85,B 0,C 180,E1 -6208.372,E2 -6208.372} C_VEL
LIN {X 0,Y 494.898,Z 406.531,A -85,B 0,C 180,E1 -6210,E2 -6210} C_VEL
LIN {X 0,Y 494.961,Z 405.713,A -85,B 0,C 180,E1 -6211.627,E2 -6211.627} C_VEL
LIN {X 0,Y 495.042,Z 403.335,A -85,B 0,C 180,E1 -6213.255,E2 -6213.255} C_VEL
LIN {X 0,Y 495.009,Z 400.414,A -85,B 0,C 180,E1 -6214.478,E2 -6214.478} C_VEL
LIN {X 0,Y 495.168,Z 395.352,A -85,B 0,C 180,E1 -6215.989,E2 -6215.989} C_VEL
LIN {X 0,Y 495.273,Z 389.367,A -85,B 0,C 180,E1 -6217.337,E2 -6217.337} C_VEL
LIN {X 0,Y 495.511,Z 382.492,A -85,B 0,C 180,E1 -6218.564,E2 -6218.564} C_VEL
LIN {X 0,Y 495.826,Z 373.889,A -85,B 0,C 180,E1 -6219.793,E2 -6219.793} C_VEL
LIN {X 0,Y 496.136,Z 365.062,A -85,B 0,C 180,E1 -6220.818,E2 -6220.818} C_VEL
LIN {X 0,Y 496.582,Z 354.197,A -85,B 0,C 180,E1 -6221.841,E2 -6221.841} C_VEL
LIN {X 0,Y 496.955,Z 342.926,A -85,B 0,C 180,E1 -6222.682,E2 -6222.682} C_VEL
LIN {X 0,Y 497.275,Z 330.934,A -85,B 0,C 180,E1 -6223.38,E2 -6223.38} C_VEL
LIN {X 0,Y 497.687,Z 317.926,A -85,B 0,C 180,E1 -6223.942,E2 -6223.942} C_VEL
LIN {X 0,Y 497.984,Z 304.659,A -85,B 0,C 180,E1 -6224.324,E2 -6224.324} C_VEL
LIN {X 0,Y 498.203,Z 284.02,A -85,B 0,C 180,E1 -6224.657,E2 -6224.657} C_VEL
LIN {X 0,Y 498.424,Z 207.401,A -85,B 0,C 180,E1 -6225.77,E2 -6225.77} C_VEL
LIN {X 0,Y 496.317,Z 194.792,A -85,B 0,C 180,E1 -6226.052,E2 -6226.052} C_VEL
LIN {X 0,Y 496.777,Z 178.009,A -85,B 0,C 180,E1 -6228.988,E2 -6228.988} C_VEL
LIN {X 0,Y 497.335,Z 162.504,A -85,B 0,C 180,E1 -6231.773,E2 -6231.773} C_VEL
LIN {X 0,Y 497.141,Z 158.921,A -85,B 0,C 180,E1 -6232.438,E2 -6232.438} C_VEL
LIN {X 0,Y 495.768,Z 151.885,A -85,B 0,C 180,E1 -6233.828,E2 -6233.828} C_VEL
LIN {X 0,Y 495.757,Z 151.72,A -85,B 0,C 180,E1 -6236.976,E2 -6236.976} C_VEL
LIN {X 0,Y 495.76,Z 151.726,A -85,B 0,C 180,E1 -6240.146,E2 -6240.146} C_VEL
LIN {X 0,Y 495.789,Z 151.726,A -85,B 0,C 180,E1 -6243.243,E2 -6243.243} C_VEL
LIN {X 0,Y 495.707,Z 151.734,A -85,B 0,C 180,E1 -6246.086,E2 -6246.086} C_VEL
LIN {X 0,Y 495.757,Z 151.722,A -85,B 0,C 180,E1 -6248.767,E2 -6248.767} C_VEL
LIN {X 0,Y 495.743,Z 151.729,A -85,B 0,C 180,E1 -6251.781,E2 -6251.781} C_VEL
LIN {X 0,Y 495.742,Z 151.736,A -85,B 0,C 180,E1 -6255.138,E2 -6255.138} C_VEL
LIN {X 0,Y 495.748,Z 151.728,A -85,B 0,C 180,E1 -6258.218,E2 -6258.218} C_VEL
LIN {X 0,Y 495.741,Z 151.725,A -85,B 0,C 180,E1 -6261.407,E2 -6261.407} C_VEL
LIN {X 0,Y 495.739,Z 151.719,A -85,B 0,C 180,E1 -6264.461,E2 -6264.461} C_VEL
LIN {X 0,Y 495.755,Z 151.73,A -85,B 0,C 180,E1 -6267.405,E2 -6267.405} C_VEL
LIN {X 0,Y 495.754,Z 151.726,A -85,B 0,C 180,E1 -6270.253,E2 -6270.253} C_VEL
LIN {X 0,Y 495.812,Z 151.723,A -85,B 0,C 180,E1 -6273.25,E2 -6273.25} C_VEL
LIN {X 0,Y 495.73,Z 151.731,A -85,B 0,C 180,E1 -6276.612,E2 -6276.612} C_VEL
LIN {X 0,Y 495.766,Z 151.727,A -85,B 0,C 180,E1 -6279.324,E2 -6279.324} C_VEL
LIN {X 0,Y 495.768,Z 151.72,A -85,B 0,C 180,E1 -6281.828,E2 -6281.828} C_VEL
LIN {X 0,Y 495.811,Z 151.725,A -85,B 0,C 180,E1 -6284.548,E2 -6284.548} C_VEL
LIN {X 0,Y 495.864,Z 151.71,A -85,B 0,C 180,E1 -6287.939,E2 -6287.939} C_VEL
LIN {X 0,Y 495.828,Z 151.721,A -85,B 0,C 180,E1 -6291.03,E2 -6291.03} C_VEL
LIN {X 0,Y 495.846,Z 151.714,A -85,B 0,C 180,E1 -6293.489,E2 -6293.489} C_VEL
LIN {X 0,Y 495.83,Z 151.723,A -85,B 0,C 180,E1 -6296.75,E2 -6296.75} C_VEL
LIN {X 0,Y 495.992,Z 151.698,A -85,B 0,C 180,E1 -6299.188,E2 -6299.188} C_VEL
LIN {X 0,Y 495.855,Z 151.71,A -85,B 0,C 180,E1 -6301.624,E2 -6301.624} C_VEL
LIN {X 0,Y 495.828,Z 151.715,A -85,B 0,C 180,E1 -6303.25,E2 -6303.25} C_VEL
LIN {X 0,Y 495.846,Z 151.721,A -85,B 0,C 180,E1 -6306.511,E2 -6306.511} C_VEL
LIN {X 0,Y 495.83,Z 151.712,A -85,B 0,C 180,E1 -6308.97,E2 -6308.97} C_VEL
LIN {X 0,Y 495.816,Z 151.722,A -85,B 0,C 180,E1 -6312.035,E2 -6312.035} C_VEL
LIN {X 0,Y 495.811,Z 151.715,A -85,B 0,C 180,E1 -6315.452,E2 -6315.452} C_VEL
LIN {X 0,Y 495.795,Z 151.729,A -85,B 0,C 180,E1 -6318.248,E2 -6318.248} C_VEL
LIN {X 0,Y 495.763,Z 151.725,A -85,B 0,C 180,E1 -6320.757,E2 -6320.757} C_VEL
LIN {X 0,Y 495.743,Z 151.727,A -85,B 0,C 180,E1 -6323.388,E2 -6323.388} C_VEL
LIN {X 0,Y 495.781,Z 151.731,A -85,B 0,C 180,E1 -6326.069,E2 -6326.069} C_VEL
LIN {X 0,Y 495.762,Z 151.726,A -85,B 0,C 180,E1 -6328.816,E2 -6328.816} C_VEL
LIN {X 0,Y 495.745,Z 151.732,A -85,B 0,C 180,E1 -6331.726,E2 -6331.726} C_VEL
LIN {X 0,Y 495.765,Z 151.711,A -85,B 0,C 180,E1 -6334.696,E2 -6334.696} C_VEL
LIN {X 0,Y 495.722,Z 151.728,A -85,B 0,C 180,E1 -6337.563,E2 -6337.563} C_VEL
LIN {X 0,Y 495.759,Z 151.726,A -85,B 0,C 180,E1 -6340.701,E2 -6340.701} C_VEL
LIN {X 0,Y 495.721,Z 151.728,A -85,B 0,C 180,E1 -6344.003,E2 -6344.003} C_VEL
LIN {X 0,Y 495.719,Z 151.732,A -85,B 0,C 180,E1 -6347.118,E2 -6347.118} C_VEL
LIN {X 0,Y 495.753,Z 151.725,A -85,B 0,C 180,E1 -6349.954,E2 -6349.954} C_VEL
LIN {X 0,Y 495.725,Z 151.733,A -85,B 0,C 180,E1 -6352.554,E2 -6352.554} C_VEL
LIN {X 0,Y 495.778,Z 151.723,A -85,B 0,C 180,E1 -6355.458,E2 -6355.458} C_VEL
LIN {X 0,Y 495.753,Z 151.726,A -85,B 0,C 180,E1 -6358.365,E2 -6358.365} C_VEL
LIN {X 0,Y 495.751,Z 151.729,A -85,B 0,C 180,E1 -6360.778,E2 -6360.778} C_VEL
LIN {X 0,Y 495.095,Z 151.814,A -85,B 0,C 180,E1 -6361.457,E2 -6361.457} C_VEL
LIN {X 0,Y 492.238,Z 152.168,A -85,B 0,C 180,E1 -6362.56,E2 -6362.56} C_VEL
LIN {X 0,Y 489.827,Z 152.471,A -85,B 0,C 180,E1 -6363.448,E2 -6363.448} C_VEL
LIN {X 0,Y 488.809,Z 152.599,A -85,B 0,C 180,E1 -6364.135,E2 -6364.135} C_VEL
LIN {X 0,Y 488.736,Z 152.605,A -85,B 0,C 180,E1 -6364.367,E2 -6364.367} C_VEL
LIN {X 0,Y 488.763,Z 152.711,A -85,B 0,C 180,E1 -6367.268,E2 -6367.268} C_VEL
LIN {X 0,Y 490.117,Z 160.982,A -85,B 0,C 180,E1 -6368.994,E2 -6368.994} C_VEL
LIN {X 0,Y 489.603,Z 176.87,A -85,B 0,C 180,E1 -6372.025,E2 -6372.025} C_VEL
LIN {X 0,Y 489.339,Z 186.312,A -85,B 0,C 180,E1 -6373.754,E2 -6373.754} C_VEL
LIN {X 0,Y 490.625,Z 193.437,A -85,B 0,C 180,E1 -6373.939,E2 -6373.939} C_VEL
LIN {X 0,Y 491.714,Z 200.598,A -85,B 0,C 180,E1 -6374.082,E2 -6374.082} C_VEL
LIN {X 0,Y 491.237,Z 293.951,A -85,B 0,C 180,E1 -6375.475,E2 -6375.475} C_VEL
LIN {X 0,Y 490.911,Z 307.092,A -85,B 0,C 180,E1 -6375.836,E2 -6375.836} C_VEL
LIN {X 0,Y 490.561,Z 319.177,A -85,B 0,C 180,E1 -6376.327,E2 -6376.327} C_VEL
LIN {X 0,Y 490.223,Z 330.237,A -85,B 0,C 180,E1 -6376.93,E2 -6376.93} C_VEL
LIN {X 0,Y 489.893,Z 340.98,A -85,B 0,C 180,E1 -6377.679,E2 -6377.679} C_VEL
LIN {X 0,Y 489.44,Z 351.695,A -85,B 0,C 180,E1 -6378.613,E2 -6378.613} C_VEL
LIN {X 0,Y 489.031,Z 361.338,A -85,B 0,C 180,E1 -6379.652,E2 -6379.652} C_VEL
LIN {X 0,Y 488.701,Z 369.238,A -85,B 0,C 180,E1 -6380.69,E2 -6380.69} C_VEL
LIN {X 0,Y 488.393,Z 376.964,A -85,B 0,C 180,E1 -6381.935,E2 -6381.935} C_VEL
LIN {X 0,Y 488.182,Z 384.053,A -85,B 0,C 180,E1 -6383.387,E2 -6383.387} C_VEL
LIN {X 0,Y 488.074,Z 388.778,A -85,B 0,C 180,E1 -6384.63,E2 -6384.63} C_VEL
LIN {X 0,Y 487.983,Z 392.398,A -85,B 0,C 180,E1 -6385.871,E2 -6385.871} C_VEL
LIN {X 0,Y 487.986,Z 394.269,A -85,B 0,C 180,E1 -6386.698,E2 -6386.698} C_VEL
LIN {X 0,Y 487.914,Z 395.681,A -85,B 0,C 180,E1 -6387.524,E2 -6387.524} C_VEL
LIN {X 0,Y 487.891,Z 396.683,A -85,B 0,C 180,E1 -6388.349,E2 -6388.349} C_VEL
LIN {X 0,Y 487.82,Z 397.54,A -85,B 0,C 180,E1 -6390,E2 -6390} C_VEL
LIN {X 0,Y 487.834,Z 397.354,A -85,B 0,C 180,E1 -6390.826,E2 -6390.826} C_VEL
LIN {X 0,Y 487.892,Z 396.768,A -85,B 0,C 180,E1 -6391.651,E2 -6391.651} C_VEL
LIN {X 0,Y 487.986,Z 394.439,A -85,B 0,C 180,E1 -6393.303,E2 -6393.303} C_VEL
LIN {X 0,Y 487.952,Z 391.565,A -85,B 0,C 180,E1 -6394.544,E2 -6394.544} C_VEL
LIN {X 0,Y 488.165,Z 386.638,A -85,B 0,C 180,E1 -6396.062,E2 -6396.062} C_VEL
LIN {X 0,Y 488.275,Z 380.662,A -85,B 0,C 180,E1 -6397.443,E2 -6397.443} C_VEL
LIN {X 0,Y 488.525,Z 373.857,A -85,B 0,C 180,E1 -6398.688,E2 -6398.688} C_VEL
LIN {X 0,Y 488.875,Z 365.363,A -85,B 0,C 180,E1 -6399.934,E2 -6399.934} C_VEL
LIN {X 0,Y 489.245,Z 356.628,A -85,B 0,C 180,E1 -6400.972,E2 -6400.972} C_VEL
LIN {X 0,Y 489.665,Z 345.872,A -85,B 0,C 180,E1 -6402.012,E2 -6402.012} C_VEL
LIN {X 0,Y 490.027,Z 335.052,A -85,B 0,C 180,E1 -6402.847,E2 -6402.847} C_VEL
LIN {X 0,Y 490.461,Z 322.999,A -85,B 0,C 180,E1 -6403.571,E2 -6403.571} C_VEL
LIN {X 0,Y 490.885,Z 310.339,A -85,B 0,C 180,E1 -6404.14,E2 -6404.14} C_VEL
LIN {X 0,Y 491.147,Z 297.839,A -85,B 0,C 180,E1 -6404.528,E2 -6404.528} C_VEL
LIN {X 0,Y 491.28,Z 281.884,A -85,B 0,C 180,E1 -6404.816,E2 -6404.816} C_VEL
LIN {X 0,Y 491.591,Z 199.147,A -85,B 0,C 180,E1 -6406.035,E2 -6406.035} C_VEL
LIN {X 0,Y 489.376,Z 186.776,A -85,B 0,C 180,E1 -6406.309,E2 -6406.309} C_VEL
LIN {X 0,Y 489.335,Z 186.118,A -85,B 0,C 180,E1 -6406.355,E2 -6406.355} C_VEL
LIN {X 0,Y 489.844,Z 169.388,A -85,B 0,C 180,E1 -6409.486,E2 -6409.486} C_VEL
LIN {X 0,Y 490.108,Z 160.266,A -85,B 0,C 180,E1 -6411.238,E2 -6411.238} C_VEL
LIN {X 0,Y 488.801,Z 153.002,A -85,B 0,C 180,E1 -6412.731,E2 -6412.731} C_VEL
LIN {X 0,Y 488.712,Z 152.611,A -85,B 0,C 180,E1 -6413.02,E2 -6413.02} C_VEL
LIN {X 0,Y 488.749,Z 152.604,A -85,B 0,C 180,E1 -6415.555,E2 -6415.555} C_VEL
LIN {X 0,Y 488.745,Z 152.605,A -85,B 0,C 180,E1 -6418.328,E2 -6418.328} C_VEL
LIN {X 0,Y 488.692,Z 152.603,A -85,B 0,C 180,E1 -6421.179,E2 -6421.179} C_VEL
LIN {X 0,Y 488.734,Z 152.606,A -85,B 0,C 180,E1 -6424.112,E2 -6424.112} C_VEL
LIN {X 0,Y 488.681,Z 152.609,A -85,B 0,C 180,E1 -6427.158,E2 -6427.158} C_VEL
LIN {X 0,Y 488.717,Z 152.601,A -85,B 0,C 180,E1 -6430.344,E2 -6430.344} C_VEL
LIN {X 0,Y 488.682,Z 152.611,A -85,B 0,C 180,E1 -6433.654,E2 -6433.654} C_VEL
LIN {X 0,Y 488.68,Z 152.601,A -85,B 0,C 180,E1 -6436.345,E2 -6436.345} C_VEL
LIN {X 0,Y 488.73,Z 152.604,A -85,B 0,C 180,E1 -6439.676,E2 -6439.676} C_VEL
LIN {X 0,Y 488.678,Z 152.604,A -85,B 0,C 180,E1 -6442.841,E2 -6442.841} C_VEL
LIN {X 0,Y 488.728,Z 152.592,A -85,B 0,C 180,E1 -6445.887,E2 -6445.887} C_VEL
LIN {X 0,Y 488.687,Z 152.608,A -85,B 0,C 180,E1 -6448.82,E2 -6448.82} C_VEL
LIN {X 0,Y 488.74,Z 152.605,A -85,B 0,C 180,E1 -6451.671,E2 -6451.671} C_VEL
LIN {X 0,Y 488.721,Z 152.605,A -85,B 0,C 180,E1 -6454.443,E2 -6454.443} C_VEL
LIN {X 0,Y 488.715,Z 152.603,A -85,B 0,C 180,E1 -6457.153,E2 -6457.153} C_VEL
LIN {X 0,Y 488.718,Z 152.609,A -85,B 0,C 180,E1 -6459.81,E2 -6459.81} C_VEL
LIN {X 0,Y 488.722,Z 152.602,A -85,B 0,C 180,E1 -6462.423,E2 -6462.423} C_VEL
LIN {X 0,Y 488.755,Z 152.594,A -85,B 0,C 180,E1 -6464.999,E2 -6464.999} C_VEL
LIN {X 0,Y 488.798,Z 152.593,A -85,B 0,C 180,E1 -6468.387,E2 -6468.387} C_VEL
LIN {X 0,Y 488.81,Z 152.594,A -85,B 0,C 180,E1 -6471.733,E2 -6471.733} C_VEL
LIN {X 0,Y 488.838,Z 152.59,A -85,B 0,C 180,E1 -6474.224,E2 -6474.224} C_VEL
LIN {X 0,Y 488.951,Z 152.575,A -85,B 0,C 180,E1 -6477.529,E2 -6477.529} C_VEL
LIN {X 0,Y 488.958,Z 152.576,A -85,B 0,C 180,E1 -6480,E2 -6480} C_VEL
LIN {X 0,Y 488.95,Z 152.574,A -85,B 0,C 180,E1 -6482.471,E2 -6482.471} C_VEL
LIN {X 0,Y 488.837,Z 152.591,A -85,B 0,C 180,E1 -6485.776,E2 -6485.776} C_VEL
LIN {X 0,Y 488.777,Z 152.596,A -85,B 0,C 180,E1 -6488.267,E2 -6488.267} C_VEL
LIN {X 0,Y 488.797,Z 152.595,A -85,B 0,C 180,E1 -6491.613,E2 -6491.613} C_VEL
LIN {X 0,Y 488.754,Z 152.603,A -85,B 0,C 180,E1 -6495.001,E2 -6495.001} C_VEL
LIN {X 0,Y 488.74,Z 152.596,A -85,B 0,C 180,E1 -6498.443,E2 -6498.443} C_VEL
LIN {X 0,Y 488.7,Z 152.612,A -85,B 0,C 180,E1 -6501.071,E2 -6501.071} C_VEL
LIN {X 0,Y 488.669,Z 152.607,A -85,B 0,C 180,E1 -6503.747,E2 -6503.747} C_VEL
LIN {X 0,Y 488.785,Z 152.601,A -85,B 0,C 180,E1 -6506.944,E2 -6506.944} C_VEL
LIN {X 0,Y 488.702,Z 152.604,A -85,B 0,C 180,E1 -6510.363,E2 -6510.363} C_VEL
LIN {X 0,Y 488.724,Z 152.603,A -85,B 0,C 180,E1 -6513.484,E2 -6513.484} C_VEL
LIN {X 0,Y 488.677,Z 152.596,A -85,B 0,C 180,E1 -6516.355,E2 -6516.355} C_VEL
LIN {X 0,Y 488.696,Z 152.611,A -85,B 0,C 180,E1 -6519.255,E2 -6519.255} C_VEL
LIN {X 0,Y 488.684,Z 152.61,A -85,B 0,C 180,E1 -6522.527,E2 -6522.527} C_VEL
LIN {X 0,Y 488.698,Z 152.611,A -85,B 0,C 180,E1 -6525.198,E2 -6525.198} C_VEL
LIN {X 0,Y 488.675,Z 152.613,A -85,B 0,C 180,E1 -6528.582,E2 -6528.582} C_VEL
LIN {X 0,Y 488.674,Z 152.602,A -85,B 0,C 180,E1 -6531.8,E2 -6531.8} C_VEL
LIN {X 0,Y 488.721,Z 152.605,A -85,B 0,C 180,E1 -6535.053,E2 -6535.053} C_VEL
LIN {X 0,Y 488.702,Z 152.608,A -85,B 0,C 180,E1 -6538.047,E2 -6538.047} C_VEL
LIN {X 0,Y 488.71,Z 152.613,A -85,B 0,C 180,E1 -6540.729,E2 -6540.729} C_VEL
LIN {X 0,Y 488.715,Z 152.599,A -85,B 0,C 180,E1 -6543.526,E2 -6543.526} C_VEL
LIN {X 0,Y 488.715,Z 152.751,A -85,B 0,C 180,E1 -6545.974,E2 -6545.974} C_VEL
LIN {X 0,Y 490.368,Z 161.253,A -85,B 0,C 180,E1 -6547.679,E2 -6547.679} C_VEL
LIN {X 0,Y 489.991,Z 173.18,A -85,B 0,C 180,E1 -6549.865,E2 -6549.865} C_VEL
LIN {X 0,Y 489.482,Z 188.675,A -85,B 0,C 180,E1 -6552.667,E2 -6552.667} C_VEL
LIN {X 0,Y 489.34,Z 194.532,A -85,B 0,C 180,E1 -6553.693,E2 -6553.693} C_VEL
LIN {X 0,Y 489.921,Z 198.512,A -85,B 0,C 180,E1 -6553.816,E2 -6553.816} C_VEL
LIN {X 0,Y 491.772,Z 209.906,A -85,B 0,C 180,E1 -6554.048,E2 -6554.048} C_VEL
LIN {X 0,Y 491.179,Z 302.316,A -85,B 0,C 180,E1 -6555.42,E2 -6555.42} C_VEL
LIN {X 0,Y 490.834,Z 315.583,A -85,B 0,C 180,E1 -6555.78,E2 -6555.78} C_VEL
LIN {X 0,Y 490.508,Z 327.738,A -85,B 0,C 180,E1 -6556.272,E2 -6556.272} C_VEL
LIN {X 0,Y 490.118,Z 339.767,A -85,B 0,C 180,E1 -6556.932,E2 -6556.932} C_VEL
LIN {X 0,Y 489.765,Z 350.284,A -85,B 0,C 180,E1 -6557.675,E2 -6557.675} C_VEL
LIN {X 0,Y 489.374,Z 360.929,A -85,B 0,C 180,E1 -6558.611,E2 -6558.611} C_VEL
LIN {X 0,Y 488.921,Z 370.517,A -85,B 0,C 180,E1 -6559.649,E2 -6559.649} C_VEL
LIN {X 0,Y 488.614,Z 378.375,A -85,B 0,C 180,E1 -6560.688,E2 -6560.688} C_VEL
LIN {X 0,Y 488.332,Z 386.047,A -85,B 0,C 180,E1 -6561.933,E2 -6561.933} C_VEL
LIN {X 0,Y 488.097,Z 393.118,A -85,B 0,C 180,E1 -6563.385,E2 -6563.385} C_VEL
LIN {X 0,Y 488.048,Z 397.821,A -85,B 0,C 180,E1 -6564.629,E2 -6564.629} C_VEL
LIN {X 0,Y 487.93,Z 401.412,A -85,B 0,C 180,E1 -6565.87,E2 -6565.87} C_VEL
LIN {X 0,Y 487.965,Z 403.266,A -85,B 0,C 180,E1 -6566.697,E2 -6566.697} C_VEL
LIN {X 0,Y 487.889,Z 405.646,A -85,B 0,C 180,E1 -6568.349,E2 -6568.349} C_VEL
LIN {X 0,Y 487.819,Z 406.466,A -85,B 0,C 180,E1 -6570,E2 -6570} C_VEL
LIN {X 0,Y 487.889,Z 405.648,A -85,B 0,C 180,E1 -6571.651,E2 -6571.651} C_VEL
LIN {X 0,Y 487.964,Z 403.27,A -85,B 0,C 180,E1 -6573.302,E2 -6573.302} C_VEL
LIN {X 0,Y 487.921,Z 400.349,A -85,B 0,C 180,E1 -6574.543,E2 -6574.543} C_VEL
LIN {X 0,Y 488.075,Z 396.394,A -85,B 0,C 180,E1 -6575.785,E2 -6575.785} C_VEL
LIN {X 0,Y 488.18,Z 390.31,A -85,B 0,C 180,E1 -6577.236,E2 -6577.236} C_VEL
LIN {X 0,Y 488.427,Z 383.659,A -85,B 0,C 180,E1 -6578.481,E2 -6578.481} C_VEL
LIN {X 0,Y 488.729,Z 375.404,A -85,B 0,C 180,E1 -6579.727,E2 -6579.727} C_VEL
LIN {X 0,Y 489.045,Z 366.941,A -85,B 0,C 180,E1 -6580.767,E2 -6580.767} C_VEL
LIN {X 0,Y 489.513,Z 356.48,A -85,B 0,C 180,E1 -6581.805,E2 -6581.805} C_VEL
LIN {X 0,Y 489.886,Z 345.303,A -85,B 0,C 180,E1 -6582.698,E2 -6582.698} C_VEL
LIN {X 0,Y 490.306,Z 332.855,A -85,B 0,C 180,E1 -6583.469,E2 -6583.469} C_VEL
LIN {X 0,Y 490.701,Z 320.527,A -85,B 0,C 180,E1 -6584.038,E2 -6584.038} C_VEL
LIN {X 0,Y 491.051,Z 307.876,A -85,B 0,C 180,E1 -6584.451,E2 -6584.451} C_VEL
LIN {X 0,Y 491.248,Z 294.677,A -85,B 0,C 180,E1 -6584.71,E2 -6584.71} C_VEL
LIN {X 0,Y 491.645,Z 208.452,A -85,B 0,C 180,E1 -6585.977,E2 -6585.977} C_VEL
LIN {X 0,Y 489.371,Z 194.878,A -85,B 0,C 180,E1 -6586.276,E2 -6586.276} C_VEL
LIN {X 0,Y 489.412,Z 189.862,A -85,B 0,C 180,E1 -6587.12,E2 -6587.12} C_VEL
LIN {X 0,Y 489.959,Z 174.366,A -85,B 0,C 180,E1 -6589.917,E2 -6589.917} C_VEL
LIN {X 0,Y 490.41,Z 162.438,A -85,B 0,C 180,E1 -6592.097,E2 -6592.097} C_VEL
LIN {X 0,Y 488.984,Z 154.061,A -85,B 0,C 180,E1 -6593.729,E2 -6593.729} C_VEL
LIN {X 0,Y 488.698,Z 152.632,A -85,B 0,C 180,E1 -6594.082,E2 -6594.082} C_VEL
LIN {X 0,Y 488.722,Z 152.595,A -85,B 0,C 180,E1 -6596.927,E2 -6596.927} C_VEL
LIN {X 0,Y 488.719,Z 152.603,A -85,B 0,C 180,E1 -6600.218,E2 -6600.218} C_VEL
LIN {X 0,Y 488.73,Z 152.602,A -85,B 0,C 180,E1 -6603.483,E2 -6603.483} C_VEL
LIN {X 0,Y 488.668,Z 152.611,A -85,B 0,C 180,E1 -6606.352,E2 -6606.352} C_VEL
LIN {X 0,Y 488.695,Z 152.607,A -85,B 0,C 180,E1 -6609.253,E2 -6609.253} C_VEL
LIN {X 0,Y 488.681,Z 152.609,A -85,B 0,C 180,E1 -6612.525,E2 -6612.525} C_VEL
LIN {X 0,Y 488.705,Z 152.611,A -85,B 0,C 180,E1 -6615.198,E2 -6615.198} C_VEL
LIN {X 0,Y 488.698,Z 152.607,A -85,B 0,C 180,E1 -6618.399,E2 -6618.399} C_VEL
LIN {X 0,Y 488.695,Z 152.609,A -85,B 0,C 180,E1 -6620.946,E2 -6620.946} C_VEL
LIN {X 0,Y 488.668,Z 152.597,A -85,B 0,C 180,E1 -6623.867,E2 -6623.867} C_VEL
LIN {X 0,Y 488.725,Z 152.608,A -85,B 0,C 180,E1 -6626.876,E2 -6626.876} C_VEL
LIN {X 0,Y 488.712,Z 152.602,A -85,B 0,C 180,E1 -6629.78,E2 -6629.78} C_VEL
LIN {X 0,Y 488.78,Z 152.602,A -85,B 0,C 180,E1 -6633.056,E2 -6633.056} C_VEL
LIN {X 0,Y 488.663,Z 152.607,A -85,B 0,C 180,E1 -6636.253,E2 -6636.253} C_VEL
LIN {X 0,Y 488.734,Z 152.605,A -85,B 0,C 180,E1 -6639.175,E2 -6639.175} C_VEL
LIN {X 0,Y 488.736,Z 152.596,A -85,B 0,C 180,E1 -6641.631,E2 -6641.631} C_VEL
LIN {X 0,Y 488.748,Z 152.604,A -85,B 0,C 180,E1 -6644.999,E2 -6644.999} C_VEL
LIN {X 0,Y 488.82,Z 152.592,A -85,B 0,C 180,E1 -6648.388,E2 -6648.388} C_VEL
LIN {X 0,Y 488.803,Z 152.593,A -85,B 0,C 180,E1 -6651.733,E2 -6651.733} C_VEL
LIN {X 0,Y 488.833,Z 152.591,A -85,B 0,C 180,E1 -6654.224,E2 -6654.224} C_VEL
LIN {X 0,Y 488.945,Z 152.574,A -85,B 0,C 180,E1 -6657.529,E2 -6657.529} C_VEL
LIN {X 0,Y 488.953,Z 152.576,A -85,B 0,C 180,E1 -6660,E2 -6660} C_VEL
LIN {X 0,Y 488.946,Z 152.575,A -85,B 0,C 180,E1 -6662.471,E2 -6662.471} C_VEL
LIN {X 0,Y 488.833,Z 152.59,A -85,B 0,C 180,E1 -6665.776,E2 -6665.776} C_VEL
LIN {X 0,Y 488.804,Z 152.596,A -85,B 0,C 180,E1 -6668.267,E2 -6668.267} C_VEL
LIN {X 0,Y 488.793,Z 152.593,A -85,B 0,C 180,E1 -6671.613,E2 -6671.613} C_VEL
LIN {X 0,Y 488.749,Z 152.595,A -85,B 0,C 180,E1 -6675.001,E2 -6675.001} C_VEL
LIN {X 0,Y 488.743,Z 152.607,A -85,B 0,C 180,E1 -6678.443,E2 -6678.443} C_VEL
LIN {X 0,Y 488.698,Z 152.603,A -85,B 0,C 180,E1 -6681.071,E2 -6681.071} C_VEL
LIN {X 0,Y 488.684,Z 152.608,A -85,B 0,C 180,E1 -6683.746,E2 -6683.746} C_VEL
LIN {X 0,Y 488.781,Z 152.593,A -85,B 0,C 180,E1 -6686.944,E2 -6686.944} C_VEL
LIN {X 0,Y 488.699,Z 152.611,A -85,B 0,C 180,E1 -6690.364,E2 -6690.364} C_VEL
LIN {X 0,Y 488.726,Z 152.599,A -85,B 0,C 180,E1 -6693.485,E2 -6693.485} C_VEL
LIN {X 0,Y 488.678,Z 152.605,A -85,B 0,C 180,E1 -6696.356,E2 -6696.356} C_VEL
LIN {X 0,Y 488.693,Z 152.608,A -85,B 0,C 180,E1 -6699.255,E2 -6699.255} C_VEL
LIN {X 0,Y 488.701,Z 152.608,A -85,B 0,C 180,E1 -6701.601,E2 -6701.601} C_VEL
LIN {X 0,Y 488.695,Z 152.603,A -85,B 0,C 180,E1 -6704.804,E2 -6704.804} C_VEL
LIN {X 0,Y 488.686,Z 152.611,A -85,B 0,C 180,E1 -6707.476,E2 -6707.476} C_VEL
LIN {X 0,Y 488.728,Z 152.6,A -85,B 0,C 180,E1 -6709.678,E2 -6709.678} C_VEL
LIN {X 0,Y 488.677,Z 152.61,A -85,B 0,C 180,E1 -6712.842,E2 -6712.842} C_VEL
LIN {X 0,Y 488.729,Z 152.605,A -85,B 0,C 180,E1 -6715.888,E2 -6715.888} C_VEL
LIN {X 0,Y 488.689,Z 152.604,A -85,B 0,C 180,E1 -6718.821,E2 -6718.821} C_VEL
LIN {X 0,Y 488.742,Z 152.605,A -85,B 0,C 180,E1 -6721.672,E2 -6721.672} C_VEL
LIN {X 0,Y 488.736,Z 152.605,A -85,B 0,C 180,E1 -6724.367,E2 -6724.367} C_VEL
LIN {X 0,Y 488.066,Z 152.691,A -85,B 0,C 180,E1 -6724.826,E2 -6724.826} C_VEL
LIN {X 0,Y 485.202,Z 153.047,A -85,B 0,C 180,E1 -6725.543,E2 -6725.543} C_VEL
LIN {X 0,Y 482.327,Z 153.406,A -85,B 0,C 180,E1 -6726.267,E2 -6726.267} C_VEL
LIN {X 0,Y 481.662,Z 153.487,A -85,B 0,C 180,E1 -6726.736,E2 -6726.736} C_VEL
LIN {X 0,Y 481.73,Z 153.751,A -85,B 0,C 180,E1 -6727.147,E2 -6727.147} C_VEL
LIN {X 0,Y 483.18,Z 162.146,A -85,B 0,C 180,E1 -6728.901,E2 -6728.901} C_VEL
LIN {X 0,Y 482.6,Z 178.063,A -85,B 0,C 180,E1 -6731.974,E2 -6731.974} C_VEL
LIN {X 0,Y 482.393,Z 186.438,A -85,B 0,C 180,E1 -6733.52,E2 -6733.52} C_VEL
LIN {X 0,Y 484.563,Z 198.728,A -85,B 0,C 180,E1 -6733.811,E2 -6733.811} C_VEL
LIN {X 0,Y 484.861,Z 202.107,A -85,B 0,C 180,E1 -6733.873,E2 -6733.873} C_VEL
LIN {X 0,Y 484.371,Z 294.035,A -85,B 0,C 180,E1 -6735.264,E2 -6735.264} C_VEL
LIN {X 0,Y 484.036,Z 307.169,A -85,B 0,C 180,E1 -6735.63,E2 -6735.63} C_VEL
LIN {X 0,Y 483.668,Z 319.252,A -85,B 0,C 180,E1 -6736.129,E2 -6736.129} C_VEL
LIN {X 0,Y 483.3,Z 330.57,A -85,B 0,C 180,E1 -6736.756,E2 -6736.756} C_VEL
LIN {X 0,Y 482.906,Z 342.34,A -85,B 0,C 180,E1 -6737.605,E2 -6737.605} C_VEL
LIN {X 0,Y 482.424,Z 352.832,A -85,B 0,C 180,E1 -6738.552,E2 -6738.552} C_VEL
LIN {X 0,Y 482.033,Z 361.407,A -85,B 0,C 180,E1 -6739.5,E2 -6739.5} C_VEL
LIN {X 0,Y 481.692,Z 369.306,A -85,B 0,C 180,E1 -6740.553,E2 -6740.553} C_VEL
LIN {X 0,Y 481.354,Z 377.032,A -85,B 0,C 180,E1 -6741.816,E2 -6741.816} C_VEL
LIN {X 0,Y 481.117,Z 384.12,A -85,B 0,C 180,E1 -6743.29,E2 -6743.29} C_VEL
LIN {X 0,Y 481.017,Z 388.845,A -85,B 0,C 180,E1 -6744.551,E2 -6744.551} C_VEL
LIN {X 0,Y 480.883,Z 392.464,A -85,B 0,C 180,E1 -6745.81,E2 -6745.81} C_VEL
LIN {X 0,Y 480.911,Z 394.335,A -85,B 0,C 180,E1 -6746.649,E2 -6746.649} C_VEL
LIN {X 0,Y 480.829,Z 395.746,A -85,B 0,C 180,E1 -6747.487,E2 -6747.487} C_VEL
LIN {X 0,Y 480.76,Z 397.367,A -85,B 0,C 180,E1 -6749.163,E2 -6749.163} C_VEL
LIN {X 0,Y 480.744,Z 397.605,A -85,B 0,C 180,E1 -6750,E2 -6750} C_VEL
LIN {X 0,Y 480.76,Z 397.418,A -85,B 0,C 180,E1 -6750.838,E2 -6750.838} C_VEL
LIN {X 0,Y 480.829,Z 395.863,A -85,B 0,C 180,E1 -6752.513,E2 -6752.513} C_VEL
LIN {X 0,Y 480.91,Z 394.503,A -85,B 0,C 180,E1 -6753.351,E2 -6753.351} C_VEL
LIN {X 0,Y 480.865,Z 391.629,A -85,B 0,C 180,E1 -6754.611,E2 -6754.611} C_VEL
LIN {X 0,Y 481.061,Z 387.729,A -85,B 0,C 180,E1 -6755.87,E2 -6755.87} C_VEL
LIN {X 0,Y 481.154,Z 382.701,A -85,B 0,C 180,E1 -6757.132,E2 -6757.132} C_VEL
LIN {X 0,Y 481.396,Z 376.375,A -85,B 0,C 180,E1 -6758.395,E2 -6758.395} C_VEL
LIN {X 0,Y 481.703,Z 368.455,A -85,B 0,C 180,E1 -6759.659,E2 -6759.659} C_VEL
LIN {X 0,Y 482.133,Z 358.605,A -85,B 0,C 180,E1 -6760.924,E2 -6760.924} C_VEL
LIN {X 0,Y 482.661,Z 348.276,A -85,B 0,C 180,E1 -6761.976,E2 -6761.976} C_VEL
LIN {X 0,Y 483.015,Z 337.364,A -85,B 0,C 180,E1 -6762.872,E2 -6762.872} C_VEL
LIN {X 0,Y 483.419,Z 326.862,A -85,B 0,C 180,E1 -6763.558,E2 -6763.558} C_VEL
LIN {X 0,Y 483.849,Z 314.293,A -85,B 0,C 180,E1 -6764.189,E2 -6764.189} C_VEL
LIN {X 0,Y 484.19,Z 301.71,A -85,B 0,C 180,E1 -6764.634,E2 -6764.634} C_VEL
LIN {X 0,Y 484.418,Z 288.87,A -85,B 0,C 180,E1 -6764.923,E2 -6764.923} C_VEL
LIN {X 0,Y 484.785,Z 200.113,A -85,B 0,C 180,E1 -6766.252,E2 -6766.252} C_VEL
LIN {X 0,Y 482.388,Z 186.497,A -85,B 0,C 180,E1 -6766.567,E2 -6766.567} C_VEL
LIN {X 0,Y 482.664,Z 176.255,A -85,B 0,C 180,E1 -6768.463,E2 -6768.463} C_VEL
LIN {X 0,Y 483.157,Z 162.614,A -85,B 0,C 180,E1 -6771.101,E2 -6771.101} C_VEL
LIN {X 0,Y 481.9,Z 154.684,A -85,B 0,C 180,E1 -6772.735,E2 -6772.735} C_VEL
LIN {X 0,Y 481.667,Z 153.513,A -85,B 0,C 180,E1 -6773.06,E2 -6773.06} C_VEL
LIN {X 0,Y 481.703,Z 153.484,A -85,B 0,C 180,E1 -6775.957,E2 -6775.957} C_VEL
LIN {X 0,Y 481.7,Z 153.482,A -85,B 0,C 180,E1 -6778.781,E2 -6778.781} C_VEL
LIN {X 0,Y 481.657,Z 153.486,A -85,B 0,C 180,E1 -6782.189,E2 -6782.189} C_VEL
LIN {X 0,Y 481.692,Z 153.476,A -85,B 0,C 180,E1 -6784.681,E2 -6784.681} C_VEL
LIN {X 0,Y 481.654,Z 153.49,A -85,B 0,C 180,E1 -6788.007,E2 -6788.007} C_VEL
LIN {X 0,Y 481.655,Z 153.479,A -85,B 0,C 180,E1 -6791.041,E2 -6791.041} C_VEL
LIN {X 0,Y 481.652,Z 153.485,A -85,B 0,C 180,E1 -6794.457,E2 -6794.457} C_VEL
LIN {X 0,Y 481.644,Z 153.478,A -85,B 0,C 180,E1 -6797.839,E2 -6797.839} C_VEL
LIN {X 0,Y 481.677,Z 153.483,A -85,B 0,C 180,E1 -6800.651,E2 -6800.651} C_VEL
LIN {X 0,Y 481.626,Z 153.483,A -85,B 0,C 180,E1 -6803.375,E2 -6803.375} C_VEL
LIN {X 0,Y 481.706,Z 153.475,A -85,B 0,C 180,E1 -6806.329,E2 -6806.329} C_VEL
LIN {X 0,Y 481.645,Z 153.487,A -85,B 0,C 180,E1 -6809.417,E2 -6809.417} C_VEL
LIN {X 0,Y 481.695,Z 153.479,A -85,B 0,C 180,E1 -6812.168,E2 -6812.168} C_VEL
LIN {X 0,Y 481.686,Z 153.48,A -85,B 0,C 180,E1 -6814.968,E2 -6814.968} C_VEL
LIN {X 0,Y 481.642,Z 153.487,A -85,B 0,C 180,E1 -6817.704,E2 -6817.704} C_VEL
LIN {X 0,Y 481.698,Z 153.48,A -85,B 0,C 180,E1 -6820.393,E2 -6820.393} C_VEL
LIN {X 0,Y 481.681,Z 153.479,A -85,B 0,C 180,E1 -6823.033,E2 -6823.033} C_VEL
LIN {X 0,Y 481.682,Z 153.482,A -85,B 0,C 180,E1 -6825.638,E2 -6825.638} C_VEL
LIN {X 0,Y 481.743,Z 153.473,A -85,B 0,C 180,E1 -6828.215,E2 -6828.215} C_VEL
LIN {X 0,Y 481.755,Z 153.471,A -85,B 0,C 180,E1 -6831.611,E2 -6831.611} C_VEL
LIN {X 0,Y 481.799,Z 153.467,A -85,B 0,C 180,E1 -6834.139,E2 -6834.139} C_VEL
LIN {X 0,Y 481.918,Z 153.451,A -85,B 0,C 180,E1 -6837.492,E2 -6837.492} C_VEL
LIN {X 0,Y 481.929,Z 153.452,A -85,B 0,C 180,E1 -6840,E2 -6840} C_VEL
LIN {X 0,Y 481.917,Z 153.45,A -85,B 0,C 180,E1 -6842.507,E2 -6842.507} C_VEL
LIN {X 0,Y 481.798,Z 153.467,A -85,B 0,C 180,E1 -6845.861,E2 -6845.861} C_VEL
LIN {X 0,Y 481.732,Z 153.474,A -85,B 0,C 180,E1 -6848.389,E2 -6848.389} C_VEL
LIN {X 0,Y 481.743,Z 153.472,A -85,B 0,C 180,E1 -6851.785,E2 -6851.785} C_VEL
LIN {X 0,Y 481.735,Z 153.481,A -85,B 0,C 180,E1 -6855.224,E2 -6855.224} C_VEL
LIN {X 0,Y 481.701,Z 153.474,A -85,B 0,C 180,E1 -6858.722,E2 -6858.722} C_VEL
LIN {X 0,Y 481.638,Z 153.491,A -85,B 0,C 180,E1 -6861.395,E2 -6861.395} C_VEL
LIN {X 0,Y 481.651,Z 153.479,A -85,B 0,C 180,E1 -6864.115,E2 -6864.115} C_VEL
LIN {X 0,Y 481.74,Z 153.481,A -85,B 0,C 180,E1 -6867.139,E2 -6867.139} C_VEL
LIN {X 0,Y 481.672,Z 153.48,A -85,B 0,C 180,E1 -6869.742,E2 -6869.742} C_VEL
LIN {X 0,Y 481.665,Z 153.486,A -85,B 0,C 180,E1 -6872.675,E2 -6872.675} C_VEL
LIN {X 0,Y 481.631,Z 153.473,A -85,B 0,C 180,E1 -6875.71,E2 -6875.71} C_VEL
LIN {X 0,Y 481.666,Z 153.481,A -85,B 0,C 180,E1 -6878.86,E2 -6878.86} C_VEL
LIN {X 0,Y 481.643,Z 153.484,A -85,B 0,C 180,E1 -6881.912,E2 -6881.912} C_VEL
LIN {X 0,Y 481.65,Z 153.485,A -85,B 0,C 180,E1 -6884.459,E2 -6884.459} C_VEL
LIN {X 0,Y 481.627,Z 153.487,A -85,B 0,C 180,E1 -6887.838,E2 -6887.838} C_VEL
LIN {X 0,Y 481.666,Z 153.477,A -85,B 0,C 180,E1 -6891.141,E2 -6891.141} C_VEL
LIN {X 0,Y 481.66,Z 153.488,A -85,B 0,C 180,E1 -6894.797,E2 -6894.797} C_VEL
LIN {X 0,Y 481.671,Z 153.485,A -85,B 0,C 180,E1 -6897.326,E2 -6897.326} C_VEL
LIN {X 0,Y 481.672,Z 153.484,A -85,B 0,C 180,E1 -6900.259,E2 -6900.259} C_VEL
LIN {X 0,Y 481.686,Z 153.471,A -85,B 0,C 180,E1 -6903.109,E2 -6903.109} C_VEL
LIN {X 0,Y 481.691,Z 153.606,A -85,B 0,C 180,E1 -6905.773,E2 -6905.773} C_VEL
LIN {X 0,Y 483.389,Z 162.383,A -85,B 0,C 180,E1 -6907.564,E2 -6907.564} C_VEL
LIN {X 0,Y 483.098,Z 173.117,A -85,B 0,C 180,E1 -6909.565,E2 -6909.565} C_VEL
LIN {X 0,Y 482.484,Z 189.802,A -85,B 0,C 180,E1 -6912.626,E2 -6912.626} C_VEL
LIN {X 0,Y 482.378,Z 194.644,A -85,B 0,C 180,E1 -6913.467,E2 -6913.467} C_VEL
LIN {X 0,Y 484.108,Z 204.971,A -85,B 0,C 180,E1 -6913.715,E2 -6913.715} C_VEL
LIN {X 0,Y 484.924,Z 211.259,A -85,B 0,C 180,E1 -6913.838,E2 -6913.838} C_VEL
LIN {X 0,Y 484.328,Z 302.261,A -85,B 0,C 180,E1 -6915.209,E2 -6915.209} C_VEL
LIN {X 0,Y 483.958,Z 315.525,A -85,B 0,C 180,E1 -6915.573,E2 -6915.573} C_VEL
LIN {X 0,Y 483.618,Z 327.677,A -85,B 0,C 180,E1 -6916.073,E2 -6916.073} C_VEL
LIN {X 0,Y 483.278,Z 338.425,A -85,B 0,C 180,E1 -6916.663,E2 -6916.663} C_VEL
LIN {X 0,Y 482.832,Z 348.91,A -85,B 0,C 180,E1 -6917.389,E2 -6917.389} C_VEL
LIN {X 0,Y 482.43,Z 359.796,A -85,B 0,C 180,E1 -6918.338,E2 -6918.338} C_VEL
LIN {X 0,Y 481.98,Z 368.671,A -85,B 0,C 180,E1 -6919.285,E2 -6919.285} C_VEL
LIN {X 0,Y 481.585,Z 378.311,A -85,B 0,C 180,E1 -6920.55,E2 -6920.55} C_VEL
LIN {X 0,Y 481.276,Z 385.983,A -85,B 0,C 180,E1 -6921.814,E2 -6921.814} C_VEL
LIN {X 0,Y 481.013,Z 393.053,A -85,B 0,C 180,E1 -6923.287,E2 -6923.287} C_VEL
LIN {X 0,Y 480.964,Z 397.756,A -85,B 0,C 180,E1 -6924.55,E2 -6924.55} C_VEL
LIN {X 0,Y 480.83,Z 401.348,A -85,B 0,C 180,E1 -6925.809,E2 -6925.809} C_VEL
LIN {X 0,Y 480.889,Z 403.201,A -85,B 0,C 180,E1 -6926.648,E2 -6926.648} C_VEL
LIN {X 0,Y 480.79,Z 405.581,A -85,B 0,C 180,E1 -6928.324,E2 -6928.324} C_VEL
LIN {X 0,Y 480.743,Z 406.401,A -85,B 0,C 180,E1 -6930,E2 -6930} C_VEL
LIN {X 0,Y 480.79,Z 405.583,A -85,B 0,C 180,E1 -6931.675,E2 -6931.675} C_VEL
LIN {X 0,Y 480.888,Z 403.205,A -85,B 0,C 180,E1 -6933.351,E2 -6933.351} C_VEL
LIN {X 0,Y 480.84,Z 400.283,A -85,B 0,C 180,E1 -6934.61,E2 -6934.61} C_VEL
LIN {X 0,Y 480.995,Z 396.329,A -85,B 0,C 180,E1 -6935.87,E2 -6935.87} C_VEL
LIN {X 0,Y 481.11,Z 390.244,A -85,B 0,C 180,E1 -6937.343,E2 -6937.343} C_VEL
LIN {X 0,Y 481.37,Z 383.593,A -85,B 0,C 180,E1 -6938.606,E2 -6938.606} C_VEL
LIN {X 0,Y 481.723,Z 375.338,A -85,B 0,C 180,E1 -6939.87,E2 -6939.87} C_VEL
LIN {X 0,Y 482.053,Z 366.874,A -85,B 0,C 180,E1 -6940.925,E2 -6940.925} C_VEL
LIN {X 0,Y 482.564,Z 356.413,A -85,B 0,C 180,E1 -6941.977,E2 -6941.977} C_VEL
LIN {X 0,Y 483.002,Z 344.738,A -85,B 0,C 180,E1 -6942.919,E2 -6942.919} C_VEL
LIN {X 0,Y 483.389,Z 332.786,A -85,B 0,C 180,E1 -6943.665,E2 -6943.665} C_VEL
LIN {X 0,Y 483.827,Z 320.457,A -85,B 0,C 180,E1 -6944.242,E2 -6944.242} C_VEL
LIN {X 0,Y 484.198,Z 307.804,A -85,B 0,C 180,E1 -6944.66,E2 -6944.66} C_VEL
LIN {X 0,Y 484.38,Z 294.597,A -85,B 0,C 180,E1 -6944.923,E2 -6944.923} C_VEL
LIN {X 0,Y 484.837,Z 209.443,A -85,B 0,C 180,E1 -6946.191,E2 -6946.191} C_VEL
LIN {X 0,Y 482.379,Z 194.829,A -85,B 0,C 180,E1 -6946.517,E2 -6946.517} C_VEL
LIN {X 0,Y 482.414,Z 190.987,A -85,B 0,C 180,E1 -6947.157,E2 -6947.157} C_VEL
LIN {X 0,Y 482.988,Z 175.493,A -85,B 0,C 180,E1 -6949.995,E2 -6949.995} C_VEL
LIN {X 0,Y 483.451,Z 163.566,A -85,B 0,C 180,E1 -6952.207,E2 -6952.207} C_VEL
LIN {X 0,Y 481.689,Z 153.598,A -85,B 0,C 180,E1 -6954.226,E2 -6954.226} C_VEL
LIN {X 0,Y 481.692,Z 153.47,A -85,B 0,C 180,E1 -6957.126,E2 -6957.126} C_VEL
LIN {X 0,Y 481.669,Z 153.484,A -85,B 0,C 180,E1 -6959.741,E2 -6959.741} C_VEL
LIN {X 0,Y 481.668,Z 153.486,A -85,B 0,C 180,E1 -6962.673,E2 -6962.673} C_VEL
LIN {X 0,Y 481.627,Z 153.491,A -85,B 0,C 180,E1 -6965.709,E2 -6965.709} C_VEL
LIN {X 0,Y 481.664,Z 153.477,A -85,B 0,C 180,E1 -6968.858,E2 -6968.858} C_VEL
LIN {X 0,Y 481.639,Z 153.486,A -85,B 0,C 180,E1 -6971.911,E2 -6971.911} C_VEL
LIN {X 0,Y 481.652,Z 153.485,A -85,B 0,C 180,E1 -6974.456,E2 -6974.456} C_VEL
LIN {X 0,Y 481.64,Z 153.485,A -85,B 0,C 180,E1 -6977.838,E2 -6977.838} C_VEL
LIN {X 0,Y 481.652,Z 153.487,A -85,B 0,C 180,E1 -6980.653,E2 -6980.653} C_VEL
LIN {X 0,Y 481.618,Z 153.477,A -85,B 0,C 180,E1 -6983.375,E2 -6983.375} C_VEL
LIN {X 0,Y 481.667,Z 153.48,A -85,B 0,C 180,E1 -6986.327,E2 -6986.327} C_VEL
LIN {X 0,Y 481.638,Z 153.485,A -85,B 0,C 180,E1 -6989.417,E2 -6989.417} C_VEL
LIN {X 0,Y 481.687,Z 153.479,A -85,B 0,C 180,E1 -6992.167,E2 -6992.167} C_VEL
LIN {X 0,Y 481.68,Z 153.482,A -85,B 0,C 180,E1 -6994.968,E2 -6994.968} C_VEL
LIN {X 0,Y 481.636,Z 153.485,A -85,B 0,C 180,E1 -6997.704,E2 -6997.704} C_VEL
LIN {X 0,Y 481.692,Z 153.482,A -85,B 0,C 180,E1 -7000.392,E2 -7000.392} C_VEL
LIN {X 0,Y 481.666,Z 153.485,A -85,B 0,C 180,E1 -7003.033,E2 -7003.033} C_VEL
LIN {X 0,Y 481.675,Z 153.481,A -85,B 0,C 180,E1 -7005.638,E2 -7005.638} C_VEL
LIN {X 0,Y 481.784,Z 153.466,A -85,B 0,C 180,E1 -7008.216,E2 -7008.216} C_VEL
LIN {X 0,Y 481.749,Z 153.472,A -85,B 0,C 180,E1 -7011.611,E2 -7011.611} C_VEL
LIN {X 0,Y 481.793,Z 153.467,A -85,B 0,C 180,E1 -7014.139,E2 -7014.139} C_VEL
LIN {X 0,Y 481.913,Z 153.45,A -85,B 0,C 180,E1 -7017.493,E2 -7017.493} C_VEL
LIN {X 0,Y 481.893,Z 153.453,A -85,B 0,C 180,E1 -7020.836,E2 -7020.836} C_VEL
LIN {X 0,Y 481.913,Z 153.451,A -85,B 0,C 180,E1 -7022.508,E2 -7022.508} C_VEL
LIN {X 0,Y 481.794,Z 153.467,A -85,B 0,C 180,E1 -7025.861,E2 -7025.861} C_VEL
LIN {X 0,Y 481.75,Z 153.472,A -85,B 0,C 180,E1 -7028.389,E2 -7028.389} C_VEL
LIN {X 0,Y 481.738,Z 153.473,A -85,B 0,C 180,E1 -7031.785,E2 -7031.785} C_VEL
LIN {X 0,Y 481.73,Z 153.468,A -85,B 0,C 180,E1 -7035.225,E2 -7035.225} C_VEL
LIN {X 0,Y 481.701,Z 153.481,A -85,B 0,C 180,E1 -7038.722,E2 -7038.722} C_VEL
LIN {X 0,Y 481.638,Z 153.482,A -85,B 0,C 180,E1 -7041.395,E2 -7041.395} C_VEL
LIN {X 0,Y 481.667,Z 153.487,A -85,B 0,C 180,E1 -7044.114,E2 -7044.114} C_VEL
LIN {X 0,Y 481.736,Z 153.47,A -85,B 0,C 180,E1 -7047.14,E2 -7047.14} C_VEL
LIN {X 0,Y 481.669,Z 153.484,A -85,B 0,C 180,E1 -7049.742,E2 -7049.742} C_VEL
LIN {X 0,Y 481.662,Z 153.479,A -85,B 0,C 180,E1 -7052.675,E2 -7052.675} C_VEL
LIN {X 0,Y 481.632,Z 153.472,A -85,B 0,C 180,E1 -7055.71,E2 -7055.71} C_VEL
LIN {X 0,Y 481.662,Z 153.483,A -85,B 0,C 180,E1 -7058.86,E2 -7058.86} C_VEL
LIN {X 0,Y 481.646,Z 153.484,A -85,B 0,C 180,E1 -7061.914,E2 -7061.914} C_VEL
LIN {X 0,Y 481.648,Z 153.483,A -85,B 0,C 180,E1 -7064.459,E2 -7064.459} C_VEL
LIN {X 0,Y 481.642,Z 153.491,A -85,B 0,C 180,E1 -7067.84,E2 -7067.84} C_VEL
LIN {X 0,Y 481.656,Z 153.478,A -85,B 0,C 180,E1 -7070.655,E2 -7070.655} C_VEL
LIN {X 0,Y 481.626,Z 153.491,A -85,B 0,C 180,E1 -7073.377,E2 -7073.377} C_VEL
LIN {X 0,Y 481.707,Z 153.48,A -85,B 0,C 180,E1 -7076.331,E2 -7076.331} C_VEL
LIN {X 0,Y 481.648,Z 153.484,A -85,B 0,C 180,E1 -7079.419,E2 -7079.419} C_VEL
LIN {X 0,Y 481.698,Z 153.484,A -85,B 0,C 180,E1 -7082.169,E2 -7082.169} C_VEL
LIN {X 0,Y 481.712,Z 153.481,A -85,B 0,C 180,E1 -7084.971,E2 -7084.971} C_VEL
LIN {X 0,Y 481.662,Z 153.487,A -85,B 0,C 180,E1 -7086.736,E2 -7086.736} C_VEL
LIN {X 0,Y 481.531,Z 154.022,A -85,B 0,C 180,E1 -7087.088,E2 -7087.088} C_VEL
LIN {X 0,Y 480.817,Z 156.301,A -85,B 0,C 180,E1 -7087.627,E2 -7087.627} C_VEL
LIN {X 0,Y 476.314,Z 167.167,A -85,B 0,C 180,E1 -7089.567,E2 -7089.567} C_VEL
LIN {X 0,Y 476.003,Z 169.231,A -85,B 0,C 180,E1 -7089.97,E2 -7089.97} C_VEL
LIN {X 0,Y 475.457,Z 183.832,A -85,B 0,C 180,E1 -7092.805,E2 -7092.805} C_VEL
LIN {X 0,Y 475.451,Z 186.643,A -85,B 0,C 180,E1 -7093.283,E2 -7093.283} C_VEL
LIN {X 0,Y 478.068,Z 202.201,A -85,B 0,C 180,E1 -7093.637,E2 -7093.637} C_VEL
LIN {X 0,Y 477.516,Z 294.119,A -85,B 0,C 180,E1 -7095.048,E2 -7095.048} C_VEL
LIN {X 0,Y 477.187,Z 307.247,A -85,B 0,C 180,E1 -7095.419,E2 -7095.419} C_VEL
LIN {X 0,Y 476.774,Z 319.326,A -85,B 0,C 180,E1 -7095.924,E2 -7095.924} C_VEL
LIN {X 0,Y 476.367,Z 330.913,A -85,B 0,C 180,E1 -7096.577,E2 -7096.577} C_VEL
LIN {X 0,Y 475.978,Z 342.411,A -85,B 0,C 180,E1 -7097.421,E2 -7097.421} C_VEL
LIN {X 0,Y 475.473,Z 352.901,A -85,B 0,C 180,E1 -7098.382,E2 -7098.382} C_VEL
LIN {X 0,Y 475.033,Z 361.475,A -85,B 0,C 180,E1 -7099.343,E2 -7099.343} C_VEL
LIN {X 0,Y 474.68,Z 369.374,A -85,B 0,C 180,E1 -7100.412,E2 -7100.412} C_VEL
LIN {X 0,Y 474.303,Z 377.099,A -85,B 0,C 180,E1 -7101.694,E2 -7101.694} C_VEL
LIN {X 0,Y 474.064,Z 384.187,A -85,B 0,C 180,E1 -7103.189,E2 -7103.189} C_VEL
LIN {X 0,Y 473.96,Z 388.911,A -85,B 0,C 180,E1 -7104.47,E2 -7104.47} C_VEL
LIN {X 0,Y 473.784,Z 392.531,A -85,B 0,C 180,E1 -7105.747,E2 -7105.747} C_VEL
LIN {X 0,Y 473.837,Z 394.4,A -85,B 0,C 180,E1 -7106.599,E2 -7106.599} C_VEL
LIN {X 0,Y 473.747,Z 395.811,A -85,B 0,C 180,E1 -7107.45,E2 -7107.45} C_VEL
LIN {X 0,Y 473.689,Z 397.432,A -85,B 0,C 180,E1 -7109.15,E2 -7109.15} C_VEL
LIN {X 0,Y 473.67,Z 397.669,A -85,B 0,C 180,E1 -7110,E2 -7110} C_VEL
LIN {X 0,Y 473.689,Z 397.483,A -85,B 0,C 180,E1 -7110.85,E2 -7110.85} C_VEL
LIN {X 0,Y 473.748,Z 395.927,A -85,B 0,C 180,E1 -7112.551,E2 -7112.551} C_VEL
LIN {X 0,Y 473.836,Z 394.567,A -85,B 0,C 180,E1 -7113.402,E2 -7113.402} C_VEL
LIN {X 0,Y 473.786,Z 391.692,A -85,B 0,C 180,E1 -7114.68,E2 -7114.68} C_VEL
LIN {X 0,Y 473.984,Z 387.793,A -85,B 0,C 180,E1 -7115.958,E2 -7115.958} C_VEL
LIN {X 0,Y 474.094,Z 382.764,A -85,B 0,C 180,E1 -7117.239,E2 -7117.239} C_VEL
LIN {X 0,Y 474.346,Z 376.438,A -85,B 0,C 180,E1 -7118.521,E2 -7118.521} C_VEL
LIN {X 0,Y 474.677,Z 368.517,A -85,B 0,C 180,E1 -7119.804,E2 -7119.804} C_VEL
LIN {X 0,Y 475.154,Z 358.666,A -85,B 0,C 180,E1 -7121.086,E2 -7121.086} C_VEL
LIN {X 0,Y 475.69,Z 348.337,A -85,B 0,C 180,E1 -7122.154,E2 -7122.154} C_VEL
LIN {X 0,Y 476.121,Z 336.688,A -85,B 0,C 180,E1 -7123.117,E2 -7123.117} C_VEL
LIN {X 0,Y 476.602,Z 325.097,A -85,B 0,C 180,E1 -7123.864,E2 -7123.864} C_VEL
LIN {X 0,Y 477.038,Z 313.047,A -85,B 0,C 180,E1 -7124.45,E2 -7124.45} C_VEL
LIN {X 0,Y 477.407,Z 299.929,A -85,B 0,C 180,E1 -7124.902,E2 -7124.902} C_VEL
LIN {X 0,Y 477.581,Z 287.319,A -85,B 0,C 180,E1 -7125.169,E2 -7125.169} C_VEL
LIN {X 0,Y 478.099,Z 201.817,A -85,B 0,C 180,E1 -7126.46,E2 -7126.46} C_VEL
LIN {X 0,Y 475.435,Z 186.656,A -85,B 0,C 180,E1 -7126.811,E2 -7126.811} C_VEL
LIN {X 0,Y 475.469,Z 183.161,A -85,B 0,C 180,E1 -7127.417,E2 -7127.417} C_VEL
LIN {X 0,Y 476.18,Z 166.051,A -85,B 0,C 180,E1 -7130.745,E2 -7130.745} C_VEL
LIN {X 0,Y 475.967,Z 161.508,A -85,B 0,C 180,E1 -7131.663,E2 -7131.663} C_VEL
LIN {X 0,Y 474.663,Z 154.439,A -85,B 0,C 180,E1 -7133.206,E2 -7133.206} C_VEL
LIN {X 0,Y 474.662,Z 154.359,A -85,B 0,C 180,E1 -7136.371,E2 -7136.371} C_VEL
LIN {X 0,Y 474.622,Z 154.362,A -85,B 0,C 180,E1 -7139.252,E2 -7139.252} C_VEL
LIN {X 0,Y 474.616,Z 154.368,A -85,B 0,C 180,E1 -7142.43,E2 -7142.43} C_VEL
LIN {X 0,Y 474.619,Z 154.355,A -85,B 0,C 180,E1 -7145.469,E2 -7145.469} C_VEL
LIN {X 0,Y 474.611,Z 154.361,A -85,B 0,C 180,E1 -7148.457,E2 -7148.457} C_VEL
LIN {X 0,Y 474.619,Z 154.358,A -85,B 0,C 180,E1 -7151.785,E2 -7151.785} C_VEL
LIN {X 0,Y 474.614,Z 154.357,A -85,B 0,C 180,E1 -7155.297,E2 -7155.297} C_VEL
LIN {X 0,Y 474.618,Z 154.359,A -85,B 0,C 180,E1 -7158.214,E2 -7158.214} C_VEL
LIN {X 0,Y 474.641,Z 154.361,A -85,B 0,C 180,E1 -7160.454,E2 -7160.454} C_VEL
LIN {X 0,Y 474.588,Z 154.359,A -85,B 0,C 180,E1 -7163.676,E2 -7163.676} C_VEL
LIN {X 0,Y 474.638,Z 154.352,A -85,B 0,C 180,E1 -7166.779,E2 -7166.779} C_VEL
LIN {X 0,Y 474.6,Z 154.368,A -85,B 0,C 180,E1 -7169.769,E2 -7169.769} C_VEL
LIN {X 0,Y 474.692,Z 154.347,A -85,B 0,C 180,E1 -7172.679,E2 -7172.679} C_VEL
LIN {X 0,Y 474.633,Z 154.362,A -85,B 0,C 180,E1 -7175.506,E2 -7175.506} C_VEL
LIN {X 0,Y 474.664,Z 154.352,A -85,B 0,C 180,E1 -7179.185,E2 -7179.185} C_VEL
LIN {X 0,Y 474.649,Z 154.361,A -85,B 0,C 180,E1 -7181.884,E2 -7181.884} C_VEL
LIN {X 0,Y 474.693,Z 154.345,A -85,B 0,C 180,E1 -7184.544,E2 -7184.544} C_VEL
LIN {X 0,Y 474.697,Z 154.353,A -85,B 0,C 180,E1 -7188.037,E2 -7188.037} C_VEL
LIN {X 0,Y 474.72,Z 154.345,A -85,B 0,C 180,E1 -7191.486,E2 -7191.486} C_VEL
LIN {X 0,Y 474.761,Z 154.345,A -85,B 0,C 180,E1 -7194.052,E2 -7194.052} C_VEL
LIN {X 0,Y 474.884,Z 154.326,A -85,B 0,C 180,E1 -7197.455,E2 -7197.455} C_VEL
LIN {X 0,Y 474.901,Z 154.327,A -85,B 0,C 180,E1 -7200,E2 -7200} C_VEL
LIN {X 0,Y 474.884,Z 154.326,A -85,B 0,C 180,E1 -7202.545,E2 -7202.545} C_VEL
LIN {X 0,Y 474.761,Z 154.343,A -85,B 0,C 180,E1 -7205.948,E2 -7205.948} C_VEL
LIN {X 0,Y 474.704,Z 154.35,A -85,B 0,C 180,E1 -7208.514,E2 -7208.514} C_VEL
LIN {X 0,Y 474.697,Z 154.348,A -85,B 0,C 180,E1 -7211.963,E2 -7211.963} C_VEL
LIN {X 0,Y 474.692,Z 154.356,A -85,B 0,C 180,E1 -7215.456,E2 -7215.456} C_VEL
LIN {X 0,Y 474.656,Z 154.355,A -85,B 0,C 180,E1 -7219.011,E2 -7219.011} C_VEL
LIN {X 0,Y 474.581,Z 154.366,A -85,B 0,C 180,E1 -7221.729,E2 -7221.729} C_VEL
LIN {X 0,Y 474.632,Z 154.354,A -85,B 0,C 180,E1 -7224.494,E2 -7224.494} C_VEL
LIN {X 0,Y 474.674,Z 154.358,A -85,B 0,C 180,E1 -7227.334,E2 -7227.334} C_VEL
LIN {X 0,Y 474.597,Z 154.365,A -85,B 0,C 180,E1 -7230.81,E2 -7230.81} C_VEL
LIN {X 0,Y 474.62,Z 154.363,A -85,B 0,C 180,E1 -7233.222,E2 -7233.222} C_VEL
LIN {X 0,Y 474.584,Z 154.35,A -85,B 0,C 180,E1 -7236.324,E2 -7236.324} C_VEL
LIN {X 0,Y 474.622,Z 154.361,A -85,B 0,C 180,E1 -7239.548,E2 -7239.548} C_VEL
LIN {X 0,Y 474.596,Z 154.363,A -85,B 0,C 180,E1 -7242.234,E2 -7242.234} C_VEL
LIN {X 0,Y 474.613,Z 154.364,A -85,B 0,C 180,E1 -7245.298,E2 -7245.298} C_VEL
LIN {X 0,Y 474.602,Z 154.363,A -85,B 0,C 180,E1 -7248.213,E2 -7248.213} C_VEL
LIN {X 0,Y 474.607,Z 154.354,A -85,B 0,C 180,E1 -7251.543,E2 -7251.543} C_VEL
LIN {X 0,Y 474.621,Z 154.366,A -85,B 0,C 180,E1 -7254.726,E2 -7254.726} C_VEL
LIN {X 0,Y 474.635,Z 154.36,A -85,B 0,C 180,E1 -7257.788,E2 -7257.788} C_VEL
LIN {X 0,Y 474.607,Z 154.367,A -85,B 0,C 180,E1 -7260.889,E2 -7260.889} C_VEL
LIN {X 0,Y 474.613,Z 154.354,A -85,B 0,C 180,E1 -7263.626,E2 -7263.626} C_VEL
LIN {X 0,Y 474.634,Z 154.464,A -85,B 0,C 180,E1 -7265.564,E2 -7265.564} C_VEL
LIN {X 0,Y 476.531,Z 164.827,A -85,B 0,C 180,E1 -7267.704,E2 -7267.704} C_VEL
LIN {X 0,Y 475.882,Z 180.445,A -85,B 0,C 180,E1 -7270.637,E2 -7270.637} C_VEL
LIN {X 0,Y 475.382,Z 194.586,A -85,B 0,C 180,E1 -7273.217,E2 -7273.217} C_VEL
LIN {X 0,Y 477.495,Z 206.96,A -85,B 0,C 180,E1 -7273.514,E2 -7273.514} C_VEL
LIN {X 0,Y 478.126,Z 211.211,A -85,B 0,C 180,E1 -7273.602,E2 -7273.602} C_VEL
LIN {X 0,Y 477.471,Z 302.206,A -85,B 0,C 180,E1 -7274.991,E2 -7274.991} C_VEL
LIN {X 0,Y 477.094,Z 315.467,A -85,B 0,C 180,E1 -7275.361,E2 -7275.361} C_VEL
LIN {X 0,Y 476.716,Z 327.617,A -85,B 0,C 180,E1 -7275.867,E2 -7275.867} C_VEL
LIN {X 0,Y 476.289,Z 339.876,A -85,B 0,C 180,E1 -7276.562,E2 -7276.562} C_VEL
LIN {X 0,Y 475.819,Z 351.503,A -85,B 0,C 180,E1 -7277.421,E2 -7277.421} C_VEL
LIN {X 0,Y 475.384,Z 361.873,A -85,B 0,C 180,E1 -7278.379,E2 -7278.379} C_VEL
LIN {X 0,Y 474.9,Z 370.39,A -85,B 0,C 180,E1 -7279.34,E2 -7279.34} C_VEL
LIN {X 0,Y 474.546,Z 378.248,A -85,B 0,C 180,E1 -7280.409,E2 -7280.409} C_VEL
LIN {X 0,Y 474.236,Z 385.919,A -85,B 0,C 180,E1 -7281.692,E2 -7281.692} C_VEL
LIN {X 0,Y 473.931,Z 392.989,A -85,B 0,C 180,E1 -7283.187,E2 -7283.187} C_VEL
LIN {X 0,Y 473.883,Z 397.692,A -85,B 0,C 180,E1 -7284.468,E2 -7284.468} C_VEL
LIN {X 0,Y 473.736,Z 401.283,A -85,B 0,C 180,E1 -7285.746,E2 -7285.746} C_VEL
LIN {X 0,Y 473.796,Z 403.137,A -85,B 0,C 180,E1 -7286.598,E2 -7286.598} C_VEL
LIN {X 0,Y 473.695,Z 405.516,A -85,B 0,C 180,E1 -7288.299,E2 -7288.299} C_VEL
LIN {X 0,Y 473.688,Z 406.121,A -85,B 0,C 180,E1 -7289.15,E2 -7289.15} C_VEL
LIN {X 0,Y 473.669,Z 406.336,A -85,B 0,C 180,E1 -7290,E2 -7290} C_VEL
LIN {X 0,Y 473.688,Z 406.122,A -85,B 0,C 180,E1 -7290.85,E2 -7290.85} C_VEL
LIN {X 0,Y 473.724,Z 404.528,A -85,B 0,C 180,E1 -7292.55,E2 -7292.55} C_VEL
LIN {X 0,Y 473.796,Z 403.14,A -85,B 0,C 180,E1 -7293.401,E2 -7293.401} C_VEL
LIN {X 0,Y 473.763,Z 400.218,A -85,B 0,C 180,E1 -7294.679,E2 -7294.679} C_VEL
LIN {X 0,Y 473.882,Z 395.378,A -85,B 0,C 180,E1 -7296.2,E2 -7296.2} C_VEL
LIN {X 0,Y 474.085,Z 389.169,A -85,B 0,C 180,E1 -7297.667,E2 -7297.667} C_VEL
LIN {X 0,Y 474.39,Z 382.293,A -85,B 0,C 180,E1 -7298.948,E2 -7298.948} C_VEL
LIN {X 0,Y 474.745,Z 373.689,A -85,B 0,C 180,E1 -7300.232,E2 -7300.232} C_VEL
LIN {X 0,Y 475.189,Z 364.861,A -85,B 0,C 180,E1 -7301.301,E2 -7301.301} C_VEL
LIN {X 0,Y 475.719,Z 354.047,A -85,B 0,C 180,E1 -7302.364,E2 -7302.364} C_VEL
LIN {X 0,Y 476.153,Z 343.034,A -85,B 0,C 180,E1 -7303.224,E2 -7303.224} C_VEL
LIN {X 0,Y 476.581,Z 330.727,A -85,B 0,C 180,E1 -7303.973,E2 -7303.973} C_VEL
LIN {X 0,Y 477.073,Z 317.713,A -85,B 0,C 180,E1 -7304.557,E2 -7304.557} C_VEL
LIN {X 0,Y 477.422,Z 304.437,A -85,B 0,C 180,E1 -7304.955,E2 -7304.955} C_VEL
LIN {X 0,Y 477.63,Z 283.781,A -85,B 0,C 180,E1 -7305.303,E2 -7305.303} C_VEL
LIN {X 0,Y 478.052,Z 210.49,A -85,B 0,C 180,E1 -7306.41,E2 -7306.41} C_VEL
LIN {X 0,Y 475.42,Z 194.815,A -85,B 0,C 180,E1 -7306.763,E2 -7306.763} C_VEL
LIN {X 0,Y 475.41,Z 192.112,A -85,B 0,C 180,E1 -7307.196,E2 -7307.196} C_VEL
LIN {X 0,Y 476.032,Z 176.619,A -85,B 0,C 180,E1 -7310.074,E2 -7310.074} C_VEL
